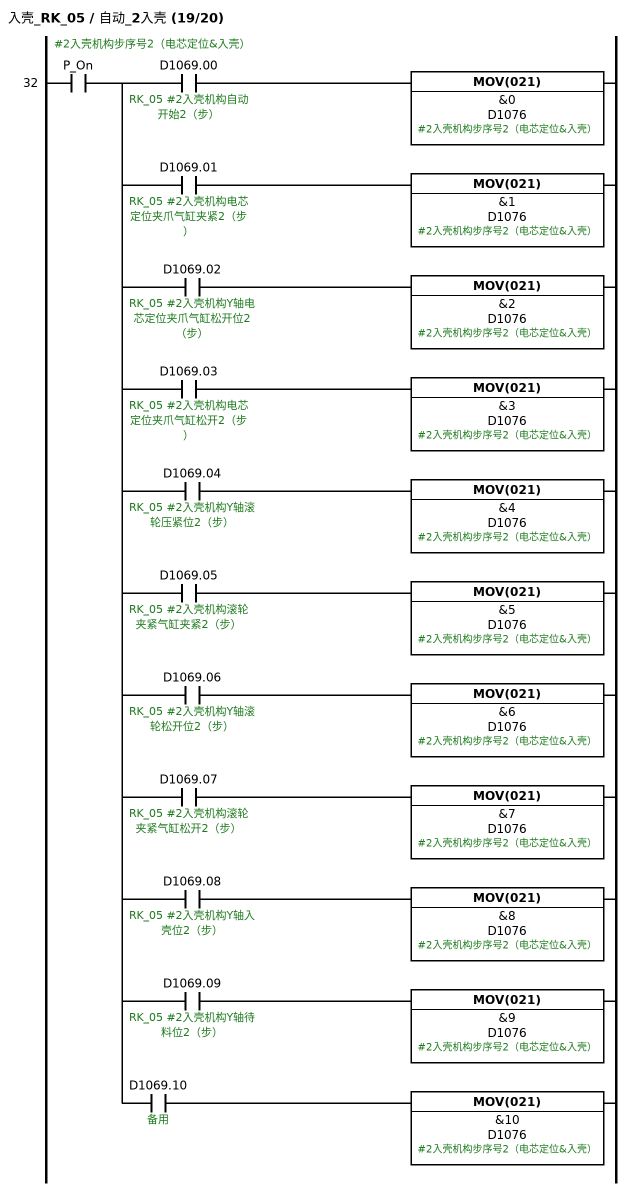
; [picture p480: 入壳_RK_05 / 自动_2入壳, rungs 32-32]
; rung 32: #2入壳机构步序号2（电芯定位&入壳）
LD P_On
OUT TR0
AND D1069.00  ; RK_05 #2入壳机构自动开始2（步）
MOV(021) &0 D1076  ; #2入壳机构步序号2（电芯定位&入壳）
LD TR0
AND D1069.01  ; RK_05 #2入壳机构电芯定位夹爪气缸夹紧2（步）
MOV(021) &1 D1076  ; #2入壳机构步序号2（电芯定位&入壳）
LD TR0
AND D1069.02  ; RK_05 #2入壳机构Y轴电芯定位夹爪气缸松开位2（步）
MOV(021) &2 D1076  ; #2入壳机构步序号2（电芯定位&入壳）
LD TR0
AND D1069.03  ; RK_05 #2入壳机构电芯定位夹爪气缸松开2（步）
MOV(021) &3 D1076  ; #2入壳机构步序号2（电芯定位&入壳）
LD TR0
AND D1069.04  ; RK_05 #2入壳机构Y轴滚轮压紧位2（步）
MOV(021) &4 D1076  ; #2入壳机构步序号2（电芯定位&入壳）
LD TR0
AND D1069.05  ; RK_05 #2入壳机构滚轮夹紧气缸夹紧2（步）
MOV(021) &5 D1076  ; #2入壳机构步序号2（电芯定位&入壳）
LD TR0
AND D1069.06  ; RK_05 #2入壳机构Y轴滚轮松开位2（步）
MOV(021) &6 D1076  ; #2入壳机构步序号2（电芯定位&入壳）
LD TR0
AND D1069.07  ; RK_05 #2入壳机构滚轮夹紧气缸松开2（步）
MOV(021) &7 D1076  ; #2入壳机构步序号2（电芯定位&入壳）
LD TR0
AND D1069.08  ; RK_05 #2入壳机构Y轴入壳位2（步）
MOV(021) &8 D1076  ; #2入壳机构步序号2（电芯定位&入壳）
LD TR0
AND D1069.09  ; RK_05 #2入壳机构Y轴待料位2（步）
MOV(021) &9 D1076  ; #2入壳机构步序号2（电芯定位&入壳）
LD TR0
AND D1069.10  ; 备用
MOV(021) &10 D1076  ; #2入壳机构步序号2（电芯定位&入壳）

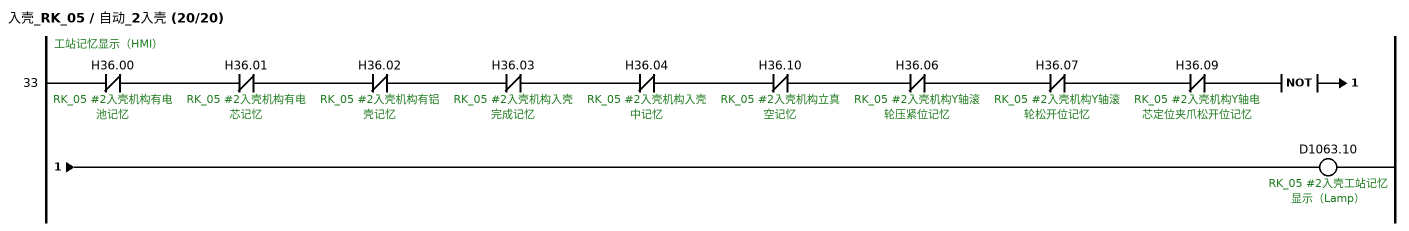
; rung 33: 工站记忆显示（HMI）
LDNOT H36.00  ; RK_05 #2入壳机构有电池记忆
ANDNOT H36.01  ; RK_05 #2入壳机构有电芯记忆
ANDNOT H36.02  ; RK_05 #2入壳机构有铝壳记忆
ANDNOT H36.03  ; RK_05 #2入壳机构入壳完成记忆
ANDNOT H36.04  ; RK_05 #2入壳机构入壳中记忆
ANDNOT H36.10  ; RK_05 #2入壳机构立真空记忆
ANDNOT H36.06  ; RK_05 #2入壳机构Y轴滚轮压紧位记忆
ANDNOT H36.07  ; RK_05 #2入壳机构Y轴滚轮松开位记忆
ANDNOT H36.09  ; RK_05 #2入壳机构Y轴电芯定位夹爪松开位记忆
NOT(520)
OUT D1063.10  ; RK_05 #2入壳工站记忆显示（Lamp）

### Section 复位

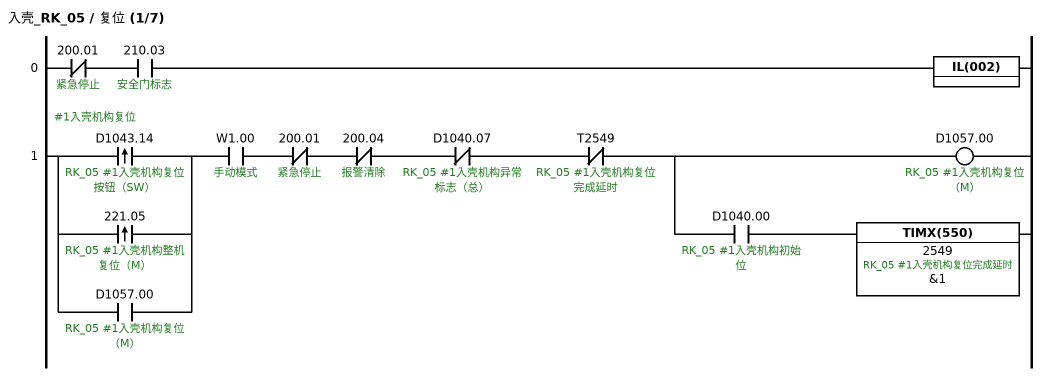
; rung 0
LDNOT 200.01  ; 紧急停止
AND 210.03  ; 安全门标志
IL(002)
; rung 1: #1入壳机构复位
@LD D1043.14  ; RK_05 #1入壳机构复位按钮（SW）
@OR 221.05  ; RK_05 #1入壳机构整机复位（M）
OR D1057.00  ; RK_05 #1入壳机构复位（M）
AND W1.00  ; 手动模式
ANDNOT 200.01  ; 紧急停止
ANDNOT 200.04  ; 报警清除
ANDNOT D1040.07  ; RK_05 #1入壳机构异常标志（总）
ANDNOT T2549  ; RK_05 #1入壳机构复位完成延时
OUT D1057.00  ; RK_05 #1入壳机构复位（M）
AND D1040.00  ; RK_05 #1入壳机构初始位
TIMX(550) 2549 &1  ; RK_05 #1入壳机构复位完成延时

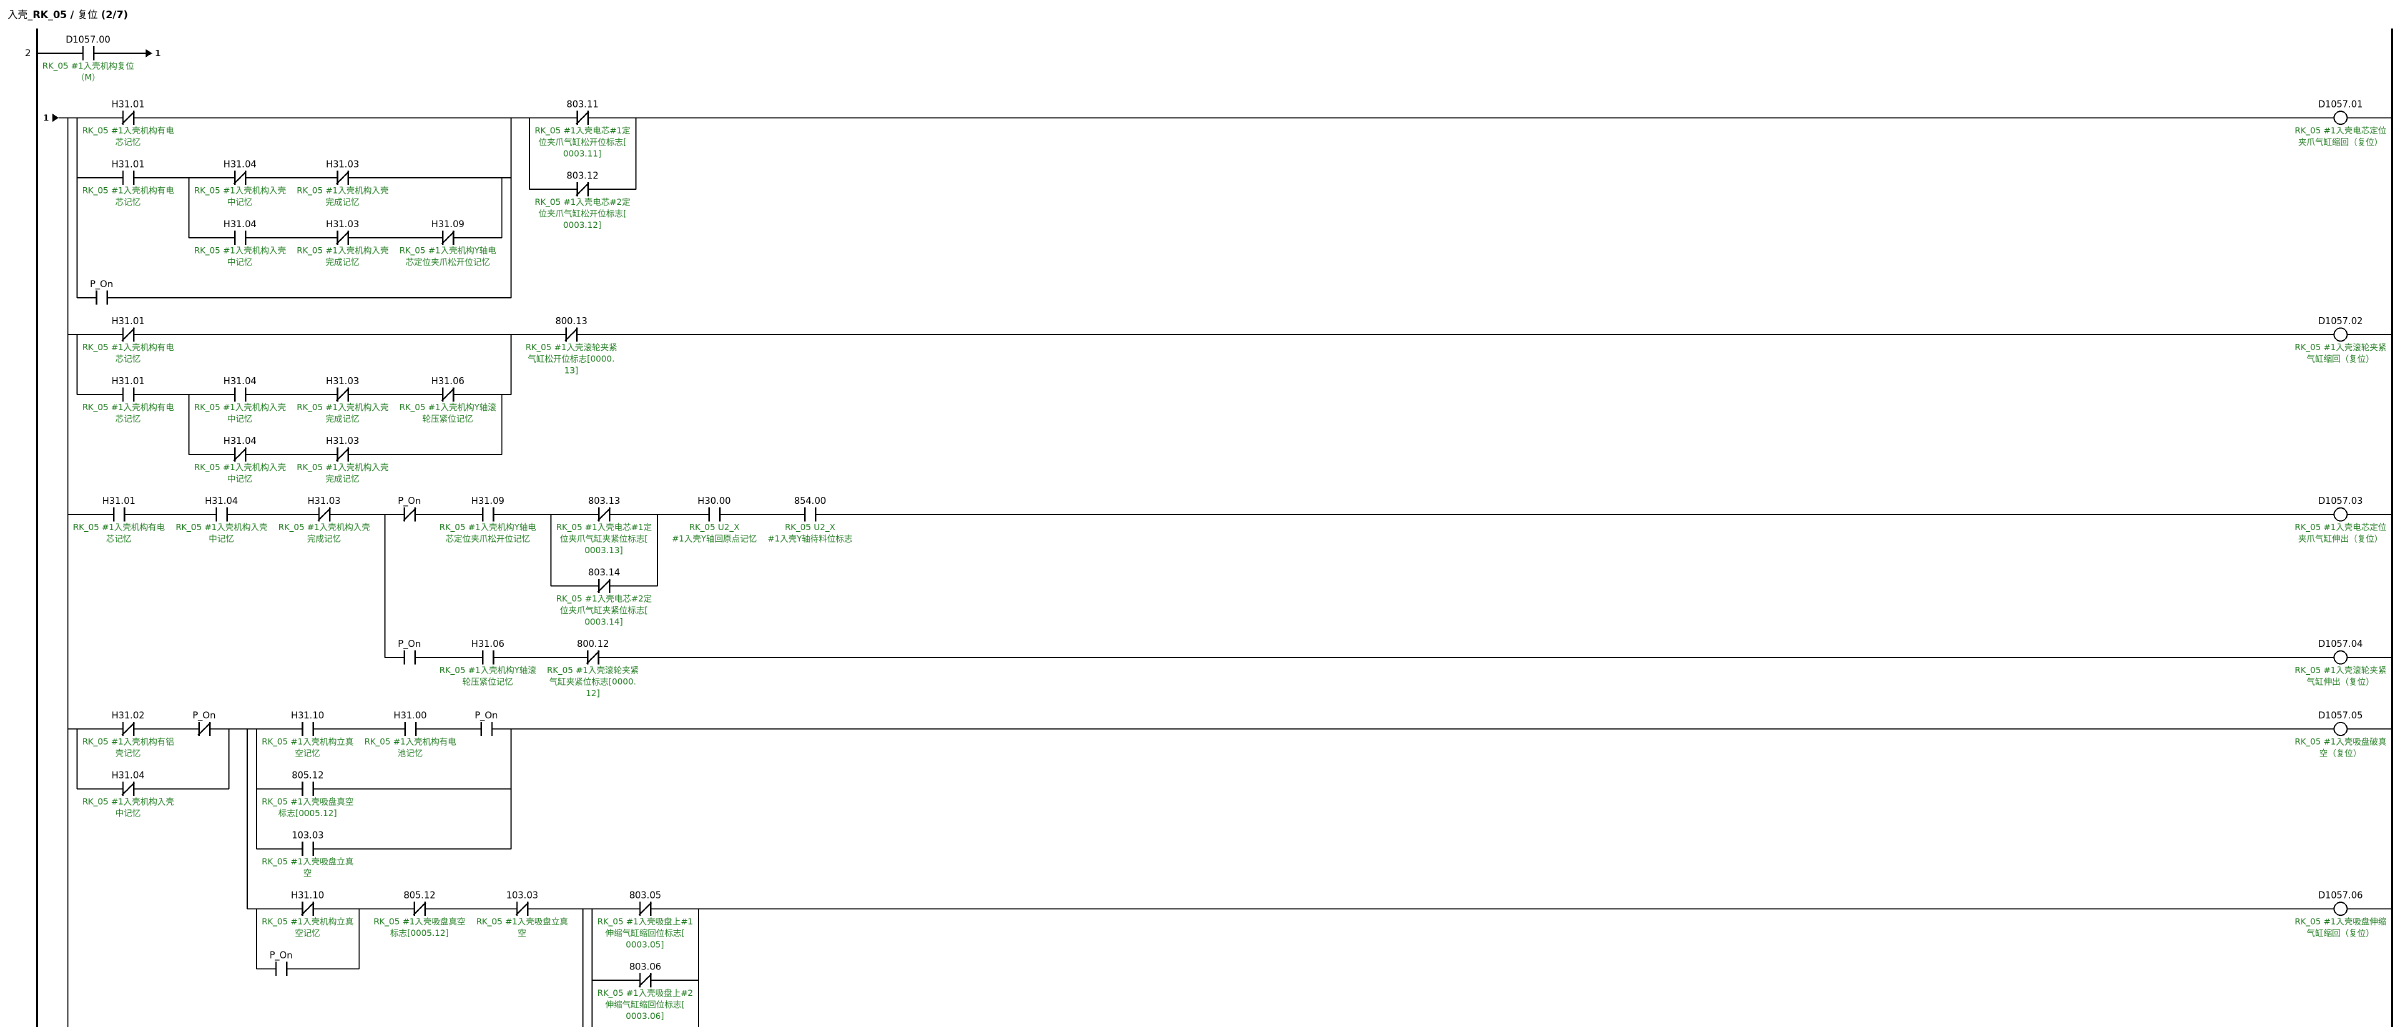

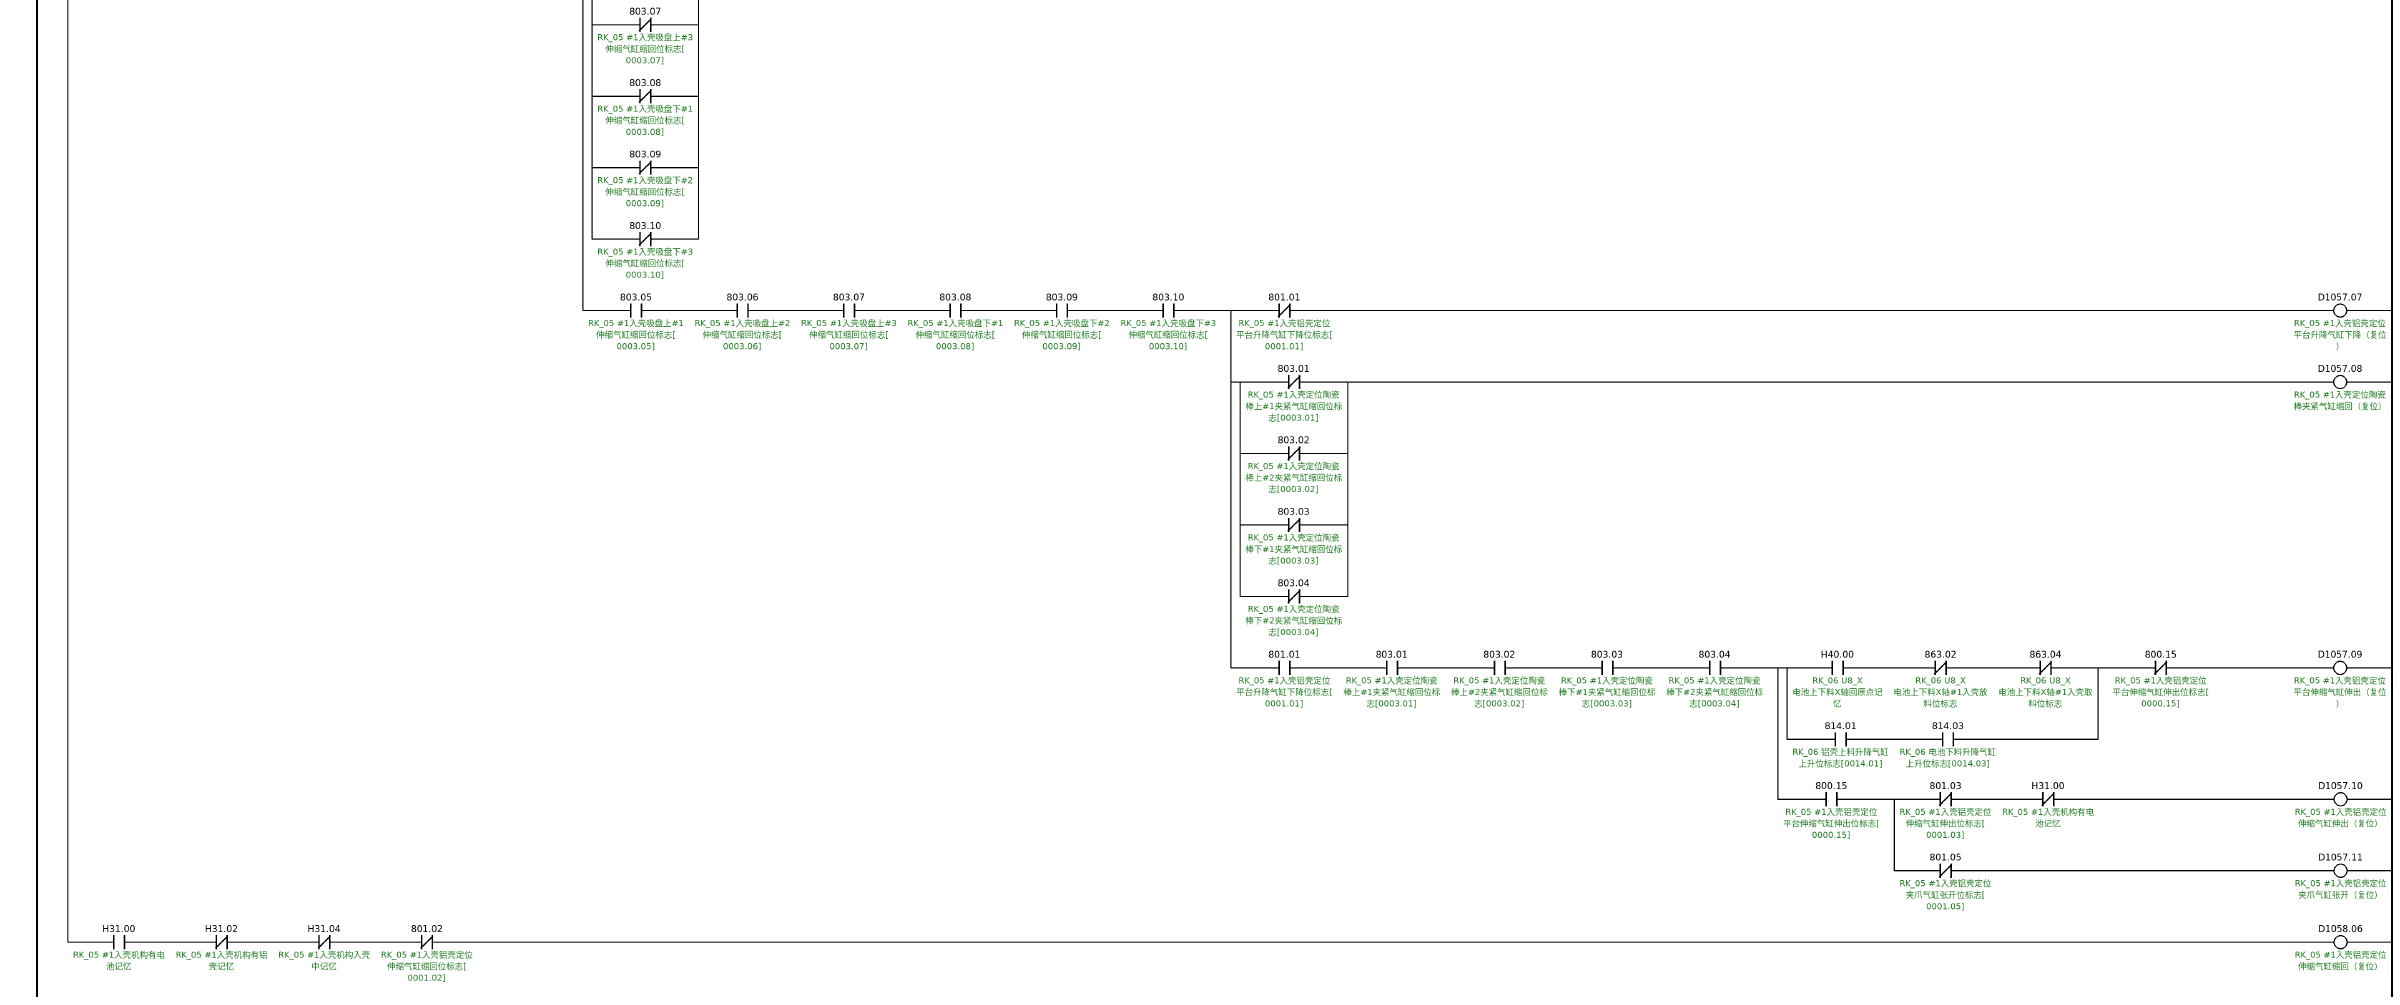
; rung 2
LD D1057.00  ; RK_05 #1入壳机构复位（M）
OUT TR0
LDNOT H31.01  ; RK_05 #1入壳机构有电芯记忆
LD H31.01  ; RK_05 #1入壳机构有电芯记忆
LDNOT H31.04  ; RK_05 #1入壳机构入壳中记忆
ANDNOT H31.03  ; RK_05 #1入壳机构入壳完成记忆
LD H31.04  ; RK_05 #1入壳机构入壳中记忆
ANDNOT H31.03  ; RK_05 #1入壳机构入壳完成记忆
ANDNOT H31.09  ; RK_05 #1入壳机构Y轴电芯定位夹爪松开位记忆
ORLD
ANDLD
ORLD
OR P_On
ANDLD
LDNOT 803.11  ; RK_05 #1入壳电芯#1定位夹爪气缸松开位标志[0003.11]
ORNOT 803.12  ; RK_05 #1入壳电芯#2定位夹爪气缸松开位标志[0003.12]
ANDLD
OUT D1057.01  ; RK_05 #1入壳电芯定位夹爪气缸缩回（复位）
LD TR0
LDNOT H31.01  ; RK_05 #1入壳机构有电芯记忆
LD H31.01  ; RK_05 #1入壳机构有电芯记忆
LD H31.04  ; RK_05 #1入壳机构入壳中记忆
ANDNOT H31.03  ; RK_05 #1入壳机构入壳完成记忆
ANDNOT H31.06  ; RK_05 #1入壳机构Y轴滚轮压紧位记忆
LDNOT H31.04  ; RK_05 #1入壳机构入壳中记忆
ANDNOT H31.03  ; RK_05 #1入壳机构入壳完成记忆
ORLD
ANDLD
ORLD
ANDLD
ANDNOT 800.13  ; RK_05 #1入壳滚轮夹紧气缸松开位标志[0000.13]
OUT D1057.02  ; RK_05 #1入壳滚轮夹紧气缸缩回（复位）
LD TR0
AND H31.01  ; RK_05 #1入壳机构有电芯记忆
AND H31.04  ; RK_05 #1入壳机构入壳中记忆
ANDNOT H31.03  ; RK_05 #1入壳机构入壳完成记忆
OUT TR1
ANDNOT P_On
AND H31.09  ; RK_05 #1入壳机构Y轴电芯定位夹爪松开位记忆
LDNOT 803.13  ; RK_05 #1入壳电芯#1定位夹爪气缸夹紧位标志[0003.13]
ORNOT 803.14  ; RK_05 #1入壳电芯#2定位夹爪气缸夹紧位标志[0003.14]
ANDLD
AND H30.00  ; RK_05 U2_X #1入壳Y轴回原点记忆
AND 854.00  ; RK_05 U2_X #1入壳Y轴待料位标志
OUT D1057.03  ; RK_05 #1入壳电芯定位夹爪气缸伸出（复位）
LD TR1
AND P_On
AND H31.06  ; RK_05 #1入壳机构Y轴滚轮压紧位记忆
ANDNOT 800.12  ; RK_05 #1入壳滚轮夹紧气缸夹紧位标志[0000.12]
OUT D1057.04  ; RK_05 #1入壳滚轮夹紧气缸伸出（复位）
LD TR0
LDNOT H31.02  ; RK_05 #1入壳机构有铝壳记忆
ANDNOT P_On
ORNOT H31.04  ; RK_05 #1入壳机构入壳中记忆
ANDLD
OUT TR1
LD H31.10  ; RK_05 #1入壳机构立真空记忆
AND H31.00  ; RK_05 #1入壳机构有电池记忆
AND P_On
OR 805.12  ; RK_05 #1入壳吸盘真空标志[0005.12]
OR 103.03  ; RK_05 #1入壳吸盘立真空
ANDLD
OUT D1057.05  ; RK_05 #1入壳吸盘破真空（复位）
LD TR1
LDNOT H31.10  ; RK_05 #1入壳机构立真空记忆
OR P_On
ANDLD
ANDNOT 805.12  ; RK_05 #1入壳吸盘真空标志[0005.12]
ANDNOT 103.03  ; RK_05 #1入壳吸盘立真空
OUT TR1
LDNOT 803.05  ; RK_05 #1入壳吸盘上#1伸缩气缸缩回位标志[0003.05]
ORNOT 803.06  ; RK_05 #1入壳吸盘上#2伸缩气缸缩回位标志[0003.06]
ORNOT 803.07  ; RK_05 #1入壳吸盘上#3伸缩气缸缩回位标志[0003.07]
ORNOT 803.08  ; RK_05 #1入壳吸盘下#1伸缩气缸缩回位标志[0003.08]
ORNOT 803.09  ; RK_05 #1入壳吸盘下#2伸缩气缸缩回位标志[0003.09]
ORNOT 803.10  ; RK_05 #1入壳吸盘下#3伸缩气缸缩回位标志[0003.10]
ANDLD
OUT D1057.06  ; RK_05 #1入壳吸盘伸缩气缸缩回（复位）
LD TR1
AND 803.05  ; RK_05 #1入壳吸盘上#1伸缩气缸缩回位标志[0003.05]
AND 803.06  ; RK_05 #1入壳吸盘上#2伸缩气缸缩回位标志[0003.06]
AND 803.07  ; RK_05 #1入壳吸盘上#3伸缩气缸缩回位标志[0003.07]
AND 803.08  ; RK_05 #1入壳吸盘下#1伸缩气缸缩回位标志[0003.08]
AND 803.09  ; RK_05 #1入壳吸盘下#2伸缩气缸缩回位标志[0003.09]
AND 803.10  ; RK_05 #1入壳吸盘下#3伸缩气缸缩回位标志[0003.10]
OUT TR1
ANDNOT 801.01  ; RK_05 #1入壳铝壳定位平台升降气缸下降位标志[0001.01]
OUT D1057.07  ; RK_05 #1入壳铝壳定位平台升降气缸下降（复位）
LD TR1
LDNOT 803.01  ; RK_05 #1入壳定位陶瓷棒上#1夹紧气缸缩回位标志[0003.01]
ORNOT 803.02  ; RK_05 #1入壳定位陶瓷棒上#2夹紧气缸缩回位标志[0003.02]
ORNOT 803.03  ; RK_05 #1入壳定位陶瓷棒下#1夹紧气缸缩回位标志[0003.03]
ORNOT 803.04  ; RK_05 #1入壳定位陶瓷棒下#2夹紧气缸缩回位标志[0003.04]
ANDLD
OUT D1057.08  ; RK_05 #1入壳定位陶瓷棒夹紧气缸缩回（复位）
LD TR1
AND 801.01  ; RK_05 #1入壳铝壳定位平台升降气缸下降位标志[0001.01]
AND 803.01  ; RK_05 #1入壳定位陶瓷棒上#1夹紧气缸缩回位标志[0003.01]
AND 803.02  ; RK_05 #1入壳定位陶瓷棒上#2夹紧气缸缩回位标志[0003.02]
AND 803.03  ; RK_05 #1入壳定位陶瓷棒下#1夹紧气缸缩回位标志[0003.03]
AND 803.04  ; RK_05 #1入壳定位陶瓷棒下#2夹紧气缸缩回位标志[0003.04]
OUT TR1
LD H40.00  ; RK_06 U8_X 电池上下料X轴回原点记忆
ANDNOT 863.02  ; RK_06 U8_X 电池上下料X轴#1入壳放料位标志
ANDNOT 863.04  ; RK_06 U8_X 电池上下料X轴#1入壳取料位标志
LD 814.01  ; RK_06 铝壳上料升降气缸上升位标志[0014.01]
AND 814.03  ; RK_06 电池下料升降气缸上升位标志[0014.03]
ORLD
ANDLD
ANDNOT 800.15  ; RK_05 #1入壳铝壳定位平台伸缩气缸伸出位标志[0000.15]
OUT D1057.09  ; RK_05 #1入壳铝壳定位平台伸缩气缸伸出（复位）
LD TR1
AND 800.15  ; RK_05 #1入壳铝壳定位平台伸缩气缸伸出位标志[0000.15]
OUT TR1
ANDNOT 801.03  ; RK_05 #1入壳铝壳定位伸缩气缸伸出位标志[0001.03]
ANDNOT H31.00  ; RK_05 #1入壳机构有电池记忆
OUT D1057.10  ; RK_05 #1入壳铝壳定位伸缩气缸伸出（复位）
LD TR1
ANDNOT 801.05  ; RK_05 #1入壳铝壳定位夹爪气缸张开位标志[0001.05]
OUT D1057.11  ; RK_05 #1入壳铝壳定位夹爪气缸张开（复位）
LD TR0
AND H31.00  ; RK_05 #1入壳机构有电池记忆
ANDNOT H31.02  ; RK_05 #1入壳机构有铝壳记忆
ANDNOT H31.04  ; RK_05 #1入壳机构入壳中记忆
ANDNOT 801.02  ; RK_05 #1入壳铝壳定位伸缩气缸缩回位标志[0001.02]
OUT D1058.06  ; RK_05 #1入壳铝壳定位伸缩气缸缩回（复位）

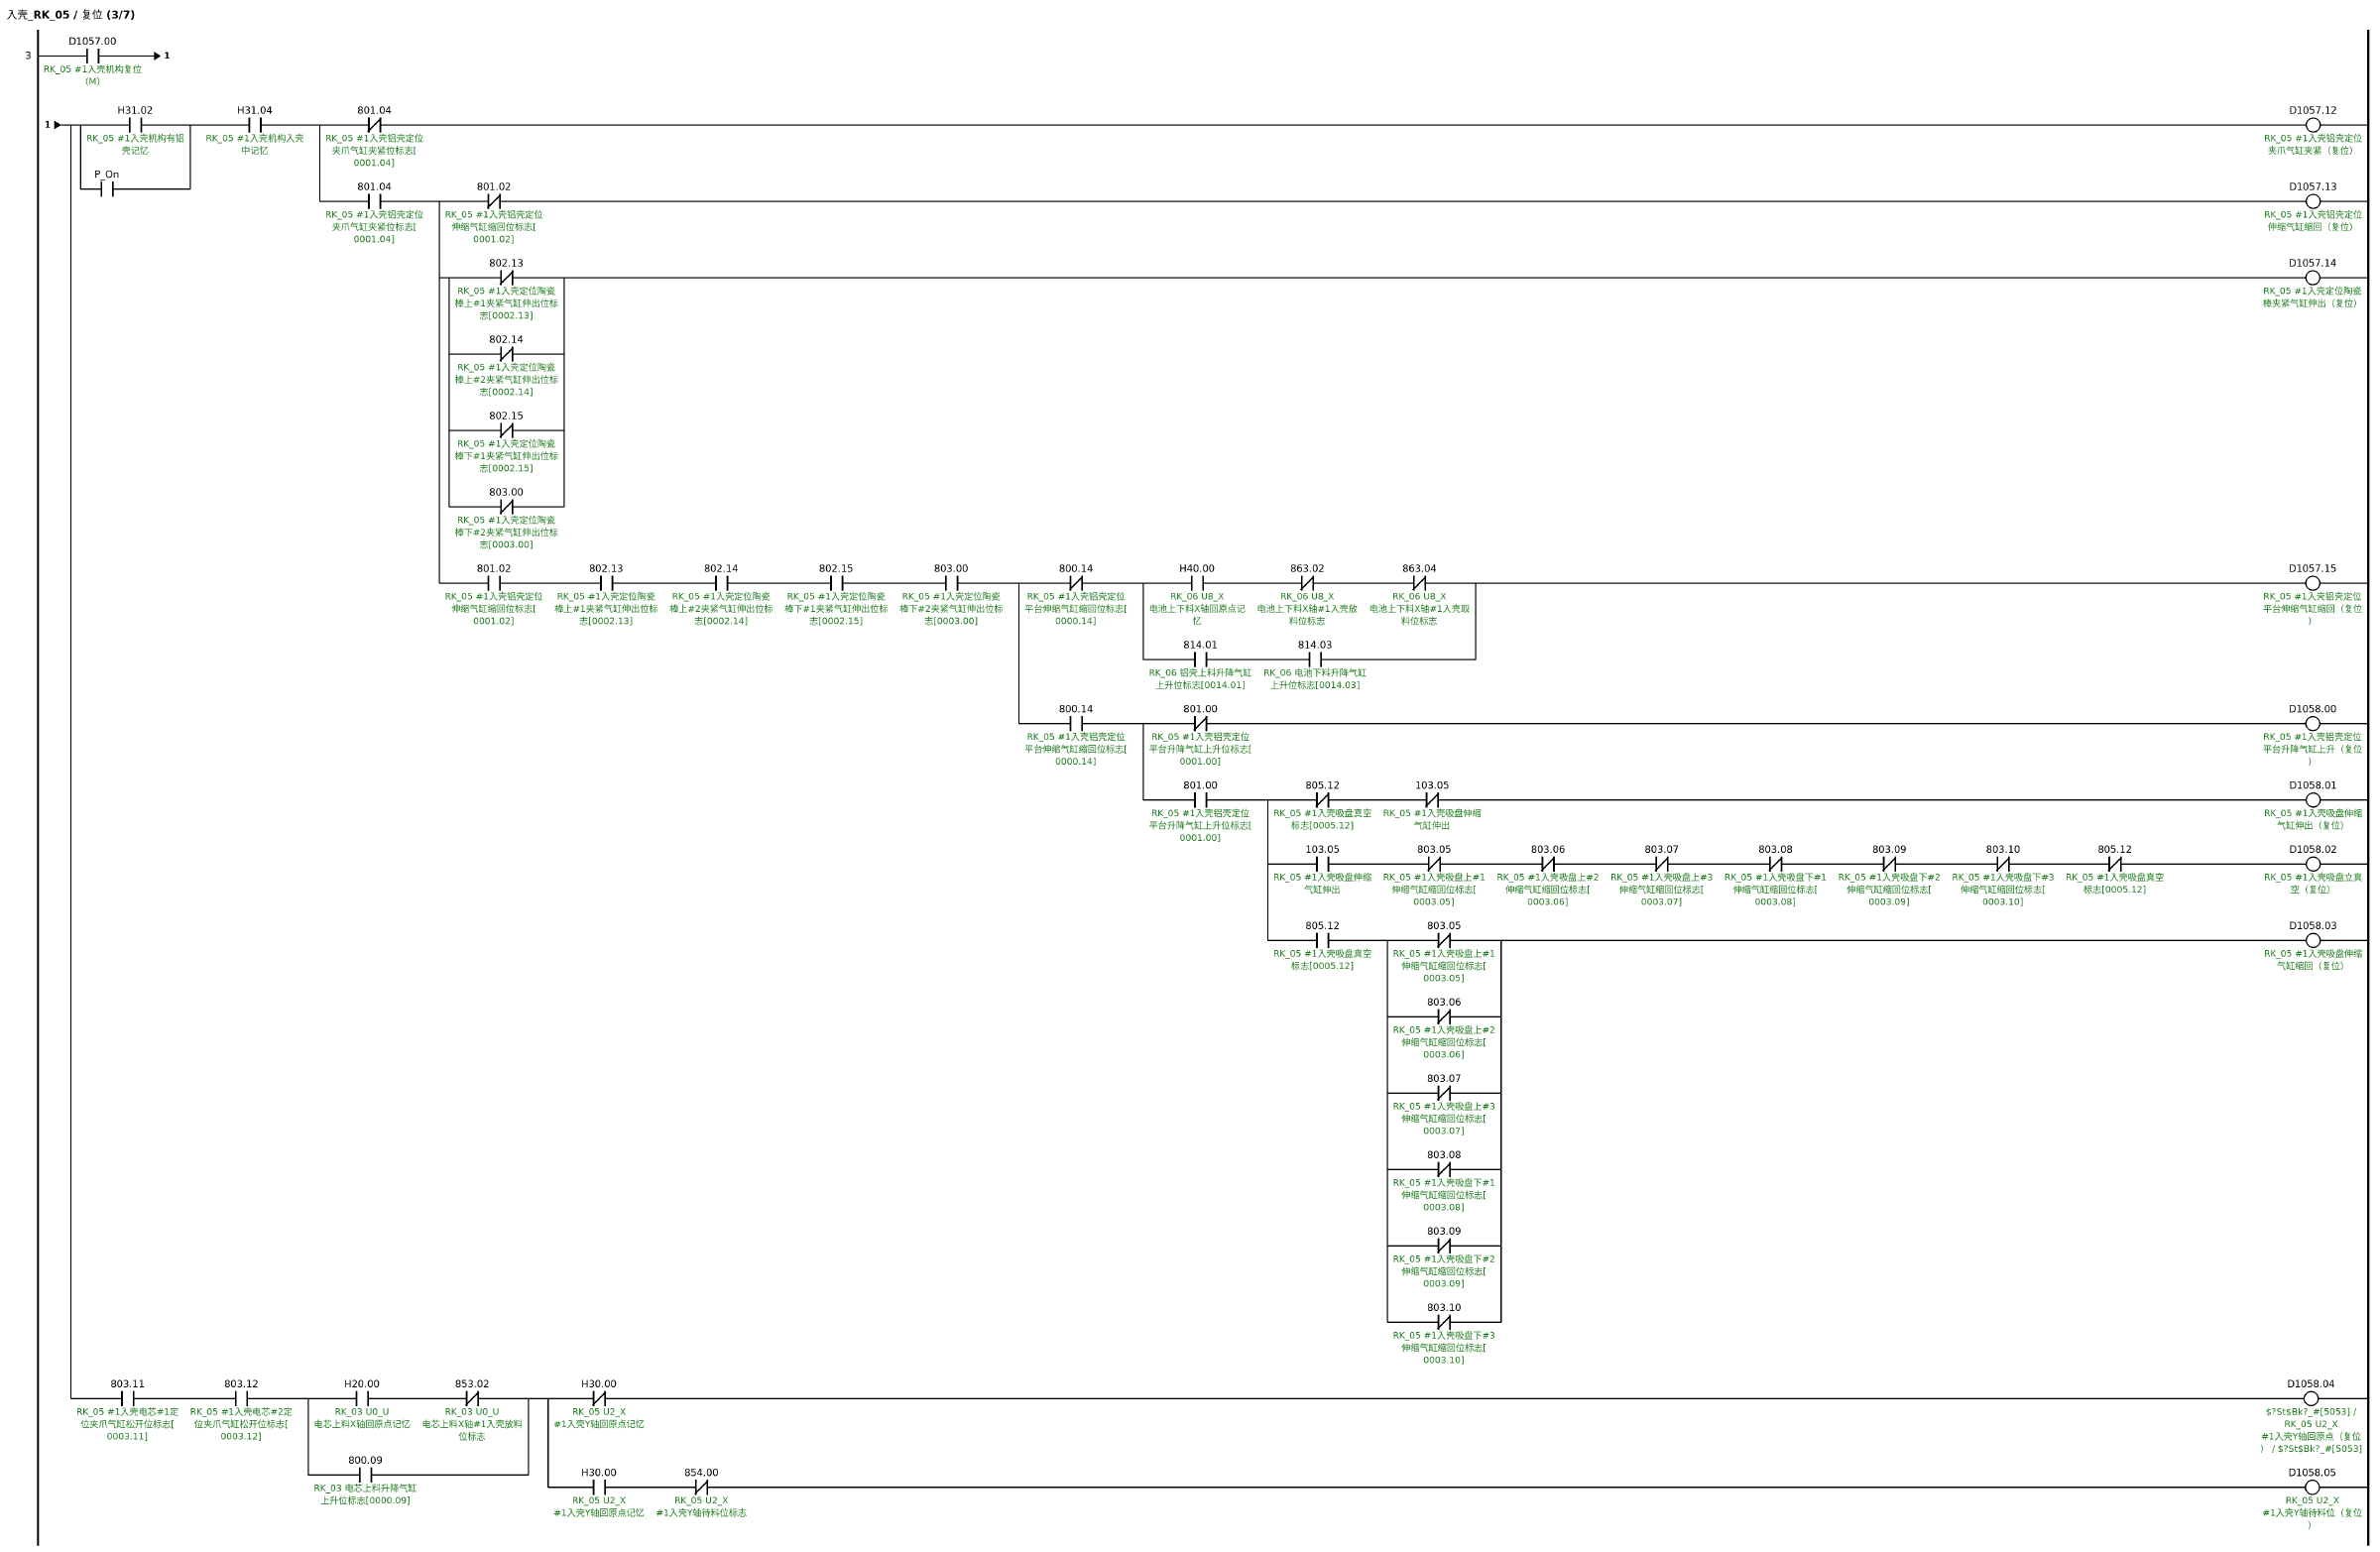
; rung 3
LD D1057.00  ; RK_05 #1入壳机构复位（M）
OUT TR0
LD H31.02  ; RK_05 #1入壳机构有铝壳记忆
OR P_On
ANDLD
AND H31.04  ; RK_05 #1入壳机构入壳中记忆
OUT TR1
ANDNOT 801.04  ; RK_05 #1入壳铝壳定位夹爪气缸夹紧位标志[0001.04]
OUT D1057.12  ; RK_05 #1入壳铝壳定位夹爪气缸夹紧（复位）
LD TR1
AND 801.04  ; RK_05 #1入壳铝壳定位夹爪气缸夹紧位标志[0001.04]
OUT TR1
ANDNOT 801.02  ; RK_05 #1入壳铝壳定位伸缩气缸缩回位标志[0001.02]
OUT D1057.13  ; RK_05 #1入壳铝壳定位伸缩气缸缩回（复位）
LD TR1
LDNOT 802.13  ; RK_05 #1入壳定位陶瓷棒上#1夹紧气缸伸出位标志[0002.13]
ORNOT 802.14  ; RK_05 #1入壳定位陶瓷棒上#2夹紧气缸伸出位标志[0002.14]
ORNOT 802.15  ; RK_05 #1入壳定位陶瓷棒下#1夹紧气缸伸出位标志[0002.15]
ORNOT 803.00  ; RK_05 #1入壳定位陶瓷棒下#2夹紧气缸伸出位标志[0003.00]
ANDLD
OUT D1057.14  ; RK_05 #1入壳定位陶瓷棒夹紧气缸伸出（复位）
LD TR1
AND 801.02  ; RK_05 #1入壳铝壳定位伸缩气缸缩回位标志[0001.02]
AND 802.13  ; RK_05 #1入壳定位陶瓷棒上#1夹紧气缸伸出位标志[0002.13]
AND 802.14  ; RK_05 #1入壳定位陶瓷棒上#2夹紧气缸伸出位标志[0002.14]
AND 802.15  ; RK_05 #1入壳定位陶瓷棒下#1夹紧气缸伸出位标志[0002.15]
AND 803.00  ; RK_05 #1入壳定位陶瓷棒下#2夹紧气缸伸出位标志[0003.00]
OUT TR1
ANDNOT 800.14  ; RK_05 #1入壳铝壳定位平台伸缩气缸缩回位标志[0000.14]
LD H40.00  ; RK_06 U8_X 电池上下料X轴回原点记忆
ANDNOT 863.02  ; RK_06 U8_X 电池上下料X轴#1入壳放料位标志
ANDNOT 863.04  ; RK_06 U8_X 电池上下料X轴#1入壳取料位标志
LD 814.01  ; RK_06 铝壳上料升降气缸上升位标志[0014.01]
AND 814.03  ; RK_06 电池下料升降气缸上升位标志[0014.03]
ORLD
ANDLD
OUT D1057.15  ; RK_05 #1入壳铝壳定位平台伸缩气缸缩回（复位）
LD TR1
AND 800.14  ; RK_05 #1入壳铝壳定位平台伸缩气缸缩回位标志[0000.14]
OUT TR1
ANDNOT 801.00  ; RK_05 #1入壳铝壳定位平台升降气缸上升位标志[0001.00]
OUT D1058.00  ; RK_05 #1入壳铝壳定位平台升降气缸上升（复位）
LD TR1
AND 801.00  ; RK_05 #1入壳铝壳定位平台升降气缸上升位标志[0001.00]
OUT TR1
ANDNOT 805.12  ; RK_05 #1入壳吸盘真空标志[0005.12]
ANDNOT 103.05  ; RK_05 #1入壳吸盘伸缩气缸伸出
OUT D1058.01  ; RK_05 #1入壳吸盘伸缩气缸伸出（复位）
LD TR1
AND 103.05  ; RK_05 #1入壳吸盘伸缩气缸伸出
ANDNOT 803.05  ; RK_05 #1入壳吸盘上#1伸缩气缸缩回位标志[0003.05]
ANDNOT 803.06  ; RK_05 #1入壳吸盘上#2伸缩气缸缩回位标志[0003.06]
ANDNOT 803.07  ; RK_05 #1入壳吸盘上#3伸缩气缸缩回位标志[0003.07]
ANDNOT 803.08  ; RK_05 #1入壳吸盘下#1伸缩气缸缩回位标志[0003.08]
ANDNOT 803.09  ; RK_05 #1入壳吸盘下#2伸缩气缸缩回位标志[0003.09]
ANDNOT 803.10  ; RK_05 #1入壳吸盘下#3伸缩气缸缩回位标志[0003.10]
ANDNOT 805.12  ; RK_05 #1入壳吸盘真空标志[0005.12]
OUT D1058.02  ; RK_05 #1入壳吸盘立真空（复位）
LD TR1
AND 805.12  ; RK_05 #1入壳吸盘真空标志[0005.12]
LDNOT 803.05  ; RK_05 #1入壳吸盘上#1伸缩气缸缩回位标志[0003.05]
ORNOT 803.06  ; RK_05 #1入壳吸盘上#2伸缩气缸缩回位标志[0003.06]
ORNOT 803.07  ; RK_05 #1入壳吸盘上#3伸缩气缸缩回位标志[0003.07]
ORNOT 803.08  ; RK_05 #1入壳吸盘下#1伸缩气缸缩回位标志[0003.08]
ORNOT 803.09  ; RK_05 #1入壳吸盘下#2伸缩气缸缩回位标志[0003.09]
ORNOT 803.10  ; RK_05 #1入壳吸盘下#3伸缩气缸缩回位标志[0003.10]
ANDLD
OUT D1058.03  ; RK_05 #1入壳吸盘伸缩气缸缩回（复位）
LD TR0
AND 803.11  ; RK_05 #1入壳电芯#1定位夹爪气缸松开位标志[0003.11]
AND 803.12  ; RK_05 #1入壳电芯#2定位夹爪气缸松开位标志[0003.12]
LD H20.00  ; RK_03 U0_U 电芯上料X轴回原点记忆
ANDNOT 853.02  ; RK_03 U0_U 电芯上料X轴#1入壳放料位标志
OR 800.09  ; RK_03 电芯上料升降气缸上升位标志[0000.09]
ANDLD
OUT TR0
ANDNOT H30.00  ; RK_05 U2_X #1入壳Y轴回原点记忆
OUT D1058.04  ; $?St$Bk?_#[5053] / RK_05 U2_X #1入壳Y轴回原点（复位） / $?St$Bk?_#[5053]
LD TR0
AND H30.00  ; RK_05 U2_X #1入壳Y轴回原点记忆
ANDNOT 854.00  ; RK_05 U2_X #1入壳Y轴待料位标志
OUT D1058.05  ; RK_05 U2_X #1入壳Y轴待料位（复位）

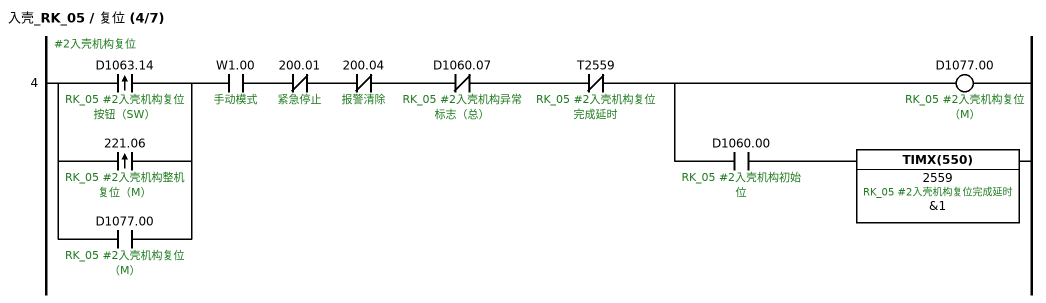
; rung 4: #2入壳机构复位
@LD D1063.14  ; RK_05 #2入壳机构复位按钮（SW）
@OR 221.06  ; RK_05 #2入壳机构整机复位（M）
OR D1077.00  ; RK_05 #2入壳机构复位（M）
AND W1.00  ; 手动模式
ANDNOT 200.01  ; 紧急停止
ANDNOT 200.04  ; 报警清除
ANDNOT D1060.07  ; RK_05 #2入壳机构异常标志（总）
ANDNOT T2559  ; RK_05 #2入壳机构复位完成延时
OUT D1077.00  ; RK_05 #2入壳机构复位（M）
AND D1060.00  ; RK_05 #2入壳机构初始位
TIMX(550) 2559 &1  ; RK_05 #2入壳机构复位完成延时

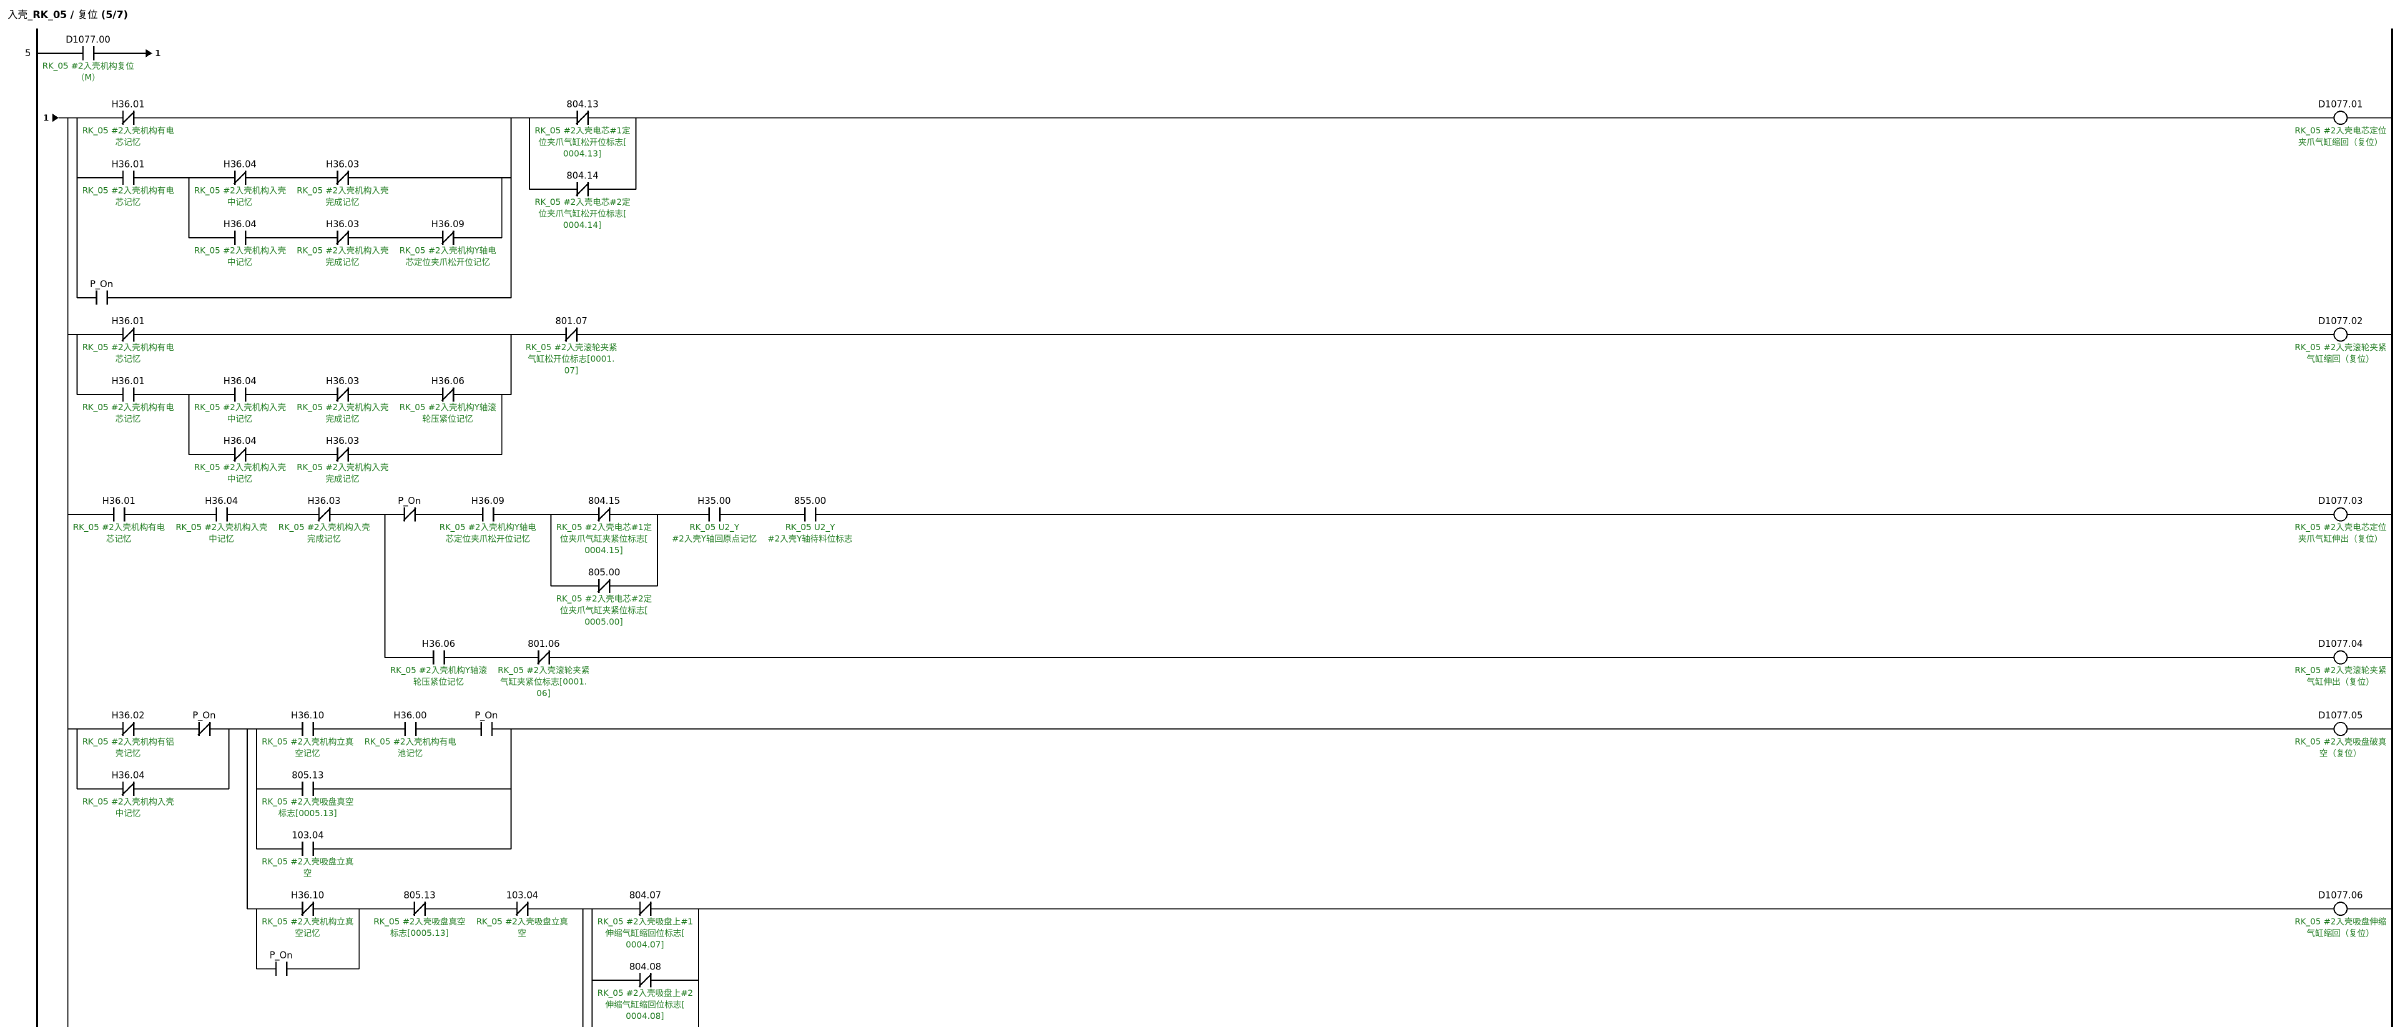

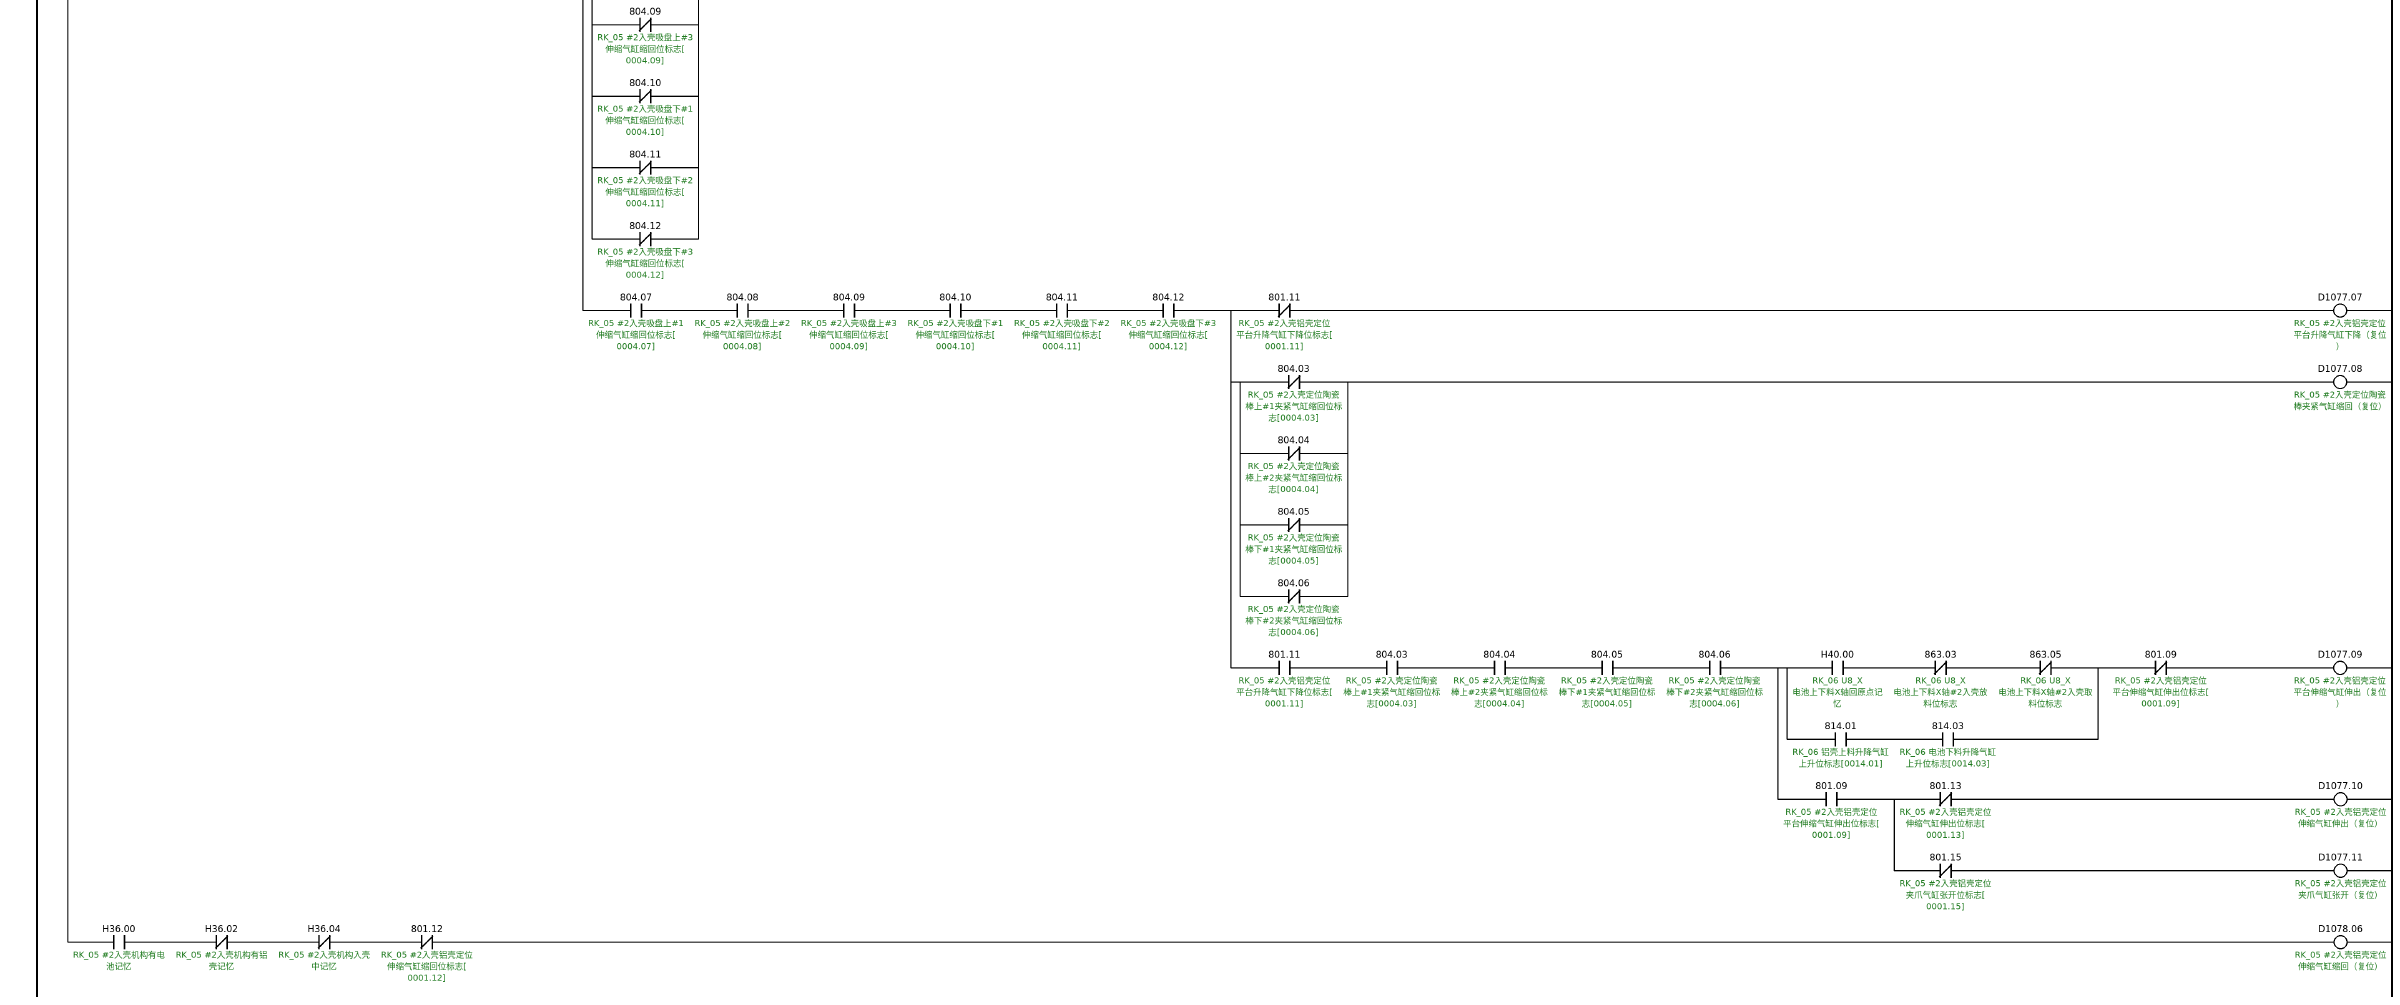
; rung 5
LD D1077.00  ; RK_05 #2入壳机构复位（M）
OUT TR0
LDNOT H36.01  ; RK_05 #2入壳机构有电芯记忆
LD H36.01  ; RK_05 #2入壳机构有电芯记忆
LDNOT H36.04  ; RK_05 #2入壳机构入壳中记忆
ANDNOT H36.03  ; RK_05 #2入壳机构入壳完成记忆
LD H36.04  ; RK_05 #2入壳机构入壳中记忆
ANDNOT H36.03  ; RK_05 #2入壳机构入壳完成记忆
ANDNOT H36.09  ; RK_05 #2入壳机构Y轴电芯定位夹爪松开位记忆
ORLD
ANDLD
ORLD
OR P_On
ANDLD
LDNOT 804.13  ; RK_05 #2入壳电芯#1定位夹爪气缸松开位标志[0004.13]
ORNOT 804.14  ; RK_05 #2入壳电芯#2定位夹爪气缸松开位标志[0004.14]
ANDLD
OUT D1077.01  ; RK_05 #2入壳电芯定位夹爪气缸缩回（复位）
LD TR0
LDNOT H36.01  ; RK_05 #2入壳机构有电芯记忆
LD H36.01  ; RK_05 #2入壳机构有电芯记忆
LD H36.04  ; RK_05 #2入壳机构入壳中记忆
ANDNOT H36.03  ; RK_05 #2入壳机构入壳完成记忆
ANDNOT H36.06  ; RK_05 #2入壳机构Y轴滚轮压紧位记忆
LDNOT H36.04  ; RK_05 #2入壳机构入壳中记忆
ANDNOT H36.03  ; RK_05 #2入壳机构入壳完成记忆
ORLD
ANDLD
ORLD
ANDLD
ANDNOT 801.07  ; RK_05 #2入壳滚轮夹紧气缸松开位标志[0001.07]
OUT D1077.02  ; RK_05 #2入壳滚轮夹紧气缸缩回（复位）
LD TR0
AND H36.01  ; RK_05 #2入壳机构有电芯记忆
AND H36.04  ; RK_05 #2入壳机构入壳中记忆
ANDNOT H36.03  ; RK_05 #2入壳机构入壳完成记忆
OUT TR1
ANDNOT P_On
AND H36.09  ; RK_05 #2入壳机构Y轴电芯定位夹爪松开位记忆
LDNOT 804.15  ; RK_05 #2入壳电芯#1定位夹爪气缸夹紧位标志[0004.15]
ORNOT 805.00  ; RK_05 #2入壳电芯#2定位夹爪气缸夹紧位标志[0005.00]
ANDLD
AND H35.00  ; RK_05 U2_Y #2入壳Y轴回原点记忆
AND 855.00  ; RK_05 U2_Y #2入壳Y轴待料位标志
OUT D1077.03  ; RK_05 #2入壳电芯定位夹爪气缸伸出（复位）
LD TR1
AND H36.06  ; RK_05 #2入壳机构Y轴滚轮压紧位记忆
ANDNOT 801.06  ; RK_05 #2入壳滚轮夹紧气缸夹紧位标志[0001.06]
OUT D1077.04  ; RK_05 #2入壳滚轮夹紧气缸伸出（复位）
LD TR0
LDNOT H36.02  ; RK_05 #2入壳机构有铝壳记忆
ANDNOT P_On
ORNOT H36.04  ; RK_05 #2入壳机构入壳中记忆
ANDLD
OUT TR1
LD H36.10  ; RK_05 #2入壳机构立真空记忆
AND H36.00  ; RK_05 #2入壳机构有电池记忆
AND P_On
OR 805.13  ; RK_05 #2入壳吸盘真空标志[0005.13]
OR 103.04  ; RK_05 #2入壳吸盘立真空
ANDLD
OUT D1077.05  ; RK_05 #2入壳吸盘破真空（复位）
LD TR1
LDNOT H36.10  ; RK_05 #2入壳机构立真空记忆
OR P_On
ANDLD
ANDNOT 805.13  ; RK_05 #2入壳吸盘真空标志[0005.13]
ANDNOT 103.04  ; RK_05 #2入壳吸盘立真空
OUT TR1
LDNOT 804.07  ; RK_05 #2入壳吸盘上#1伸缩气缸缩回位标志[0004.07]
ORNOT 804.08  ; RK_05 #2入壳吸盘上#2伸缩气缸缩回位标志[0004.08]
ORNOT 804.09  ; RK_05 #2入壳吸盘上#3伸缩气缸缩回位标志[0004.09]
ORNOT 804.10  ; RK_05 #2入壳吸盘下#1伸缩气缸缩回位标志[0004.10]
ORNOT 804.11  ; RK_05 #2入壳吸盘下#2伸缩气缸缩回位标志[0004.11]
ORNOT 804.12  ; RK_05 #2入壳吸盘下#3伸缩气缸缩回位标志[0004.12]
ANDLD
OUT D1077.06  ; RK_05 #2入壳吸盘伸缩气缸缩回（复位）
LD TR1
AND 804.07  ; RK_05 #2入壳吸盘上#1伸缩气缸缩回位标志[0004.07]
AND 804.08  ; RK_05 #2入壳吸盘上#2伸缩气缸缩回位标志[0004.08]
AND 804.09  ; RK_05 #2入壳吸盘上#3伸缩气缸缩回位标志[0004.09]
AND 804.10  ; RK_05 #2入壳吸盘下#1伸缩气缸缩回位标志[0004.10]
AND 804.11  ; RK_05 #2入壳吸盘下#2伸缩气缸缩回位标志[0004.11]
AND 804.12  ; RK_05 #2入壳吸盘下#3伸缩气缸缩回位标志[0004.12]
OUT TR1
ANDNOT 801.11  ; RK_05 #2入壳铝壳定位平台升降气缸下降位标志[0001.11]
OUT D1077.07  ; RK_05 #2入壳铝壳定位平台升降气缸下降（复位）
LD TR1
LDNOT 804.03  ; RK_05 #2入壳定位陶瓷棒上#1夹紧气缸缩回位标志[0004.03]
ORNOT 804.04  ; RK_05 #2入壳定位陶瓷棒上#2夹紧气缸缩回位标志[0004.04]
ORNOT 804.05  ; RK_05 #2入壳定位陶瓷棒下#1夹紧气缸缩回位标志[0004.05]
ORNOT 804.06  ; RK_05 #2入壳定位陶瓷棒下#2夹紧气缸缩回位标志[0004.06]
ANDLD
OUT D1077.08  ; RK_05 #2入壳定位陶瓷棒夹紧气缸缩回（复位）
LD TR1
AND 801.11  ; RK_05 #2入壳铝壳定位平台升降气缸下降位标志[0001.11]
AND 804.03  ; RK_05 #2入壳定位陶瓷棒上#1夹紧气缸缩回位标志[0004.03]
AND 804.04  ; RK_05 #2入壳定位陶瓷棒上#2夹紧气缸缩回位标志[0004.04]
AND 804.05  ; RK_05 #2入壳定位陶瓷棒下#1夹紧气缸缩回位标志[0004.05]
AND 804.06  ; RK_05 #2入壳定位陶瓷棒下#2夹紧气缸缩回位标志[0004.06]
OUT TR1
LD H40.00  ; RK_06 U8_X 电池上下料X轴回原点记忆
ANDNOT 863.03  ; RK_06 U8_X 电池上下料X轴#2入壳放料位标志
ANDNOT 863.05  ; RK_06 U8_X 电池上下料X轴#2入壳取料位标志
LD 814.01  ; RK_06 铝壳上料升降气缸上升位标志[0014.01]
AND 814.03  ; RK_06 电池下料升降气缸上升位标志[0014.03]
ORLD
ANDLD
ANDNOT 801.09  ; RK_05 #2入壳铝壳定位平台伸缩气缸伸出位标志[0001.09]
OUT D1077.09  ; RK_05 #2入壳铝壳定位平台伸缩气缸伸出（复位）
LD TR1
AND 801.09  ; RK_05 #2入壳铝壳定位平台伸缩气缸伸出位标志[0001.09]
OUT TR1
ANDNOT 801.13  ; RK_05 #2入壳铝壳定位伸缩气缸伸出位标志[0001.13]
OUT D1077.10  ; RK_05 #2入壳铝壳定位伸缩气缸伸出（复位）
LD TR1
ANDNOT 801.15  ; RK_05 #2入壳铝壳定位夹爪气缸张开位标志[0001.15]
OUT D1077.11  ; RK_05 #2入壳铝壳定位夹爪气缸张开（复位）
LD TR0
AND H36.00  ; RK_05 #2入壳机构有电池记忆
ANDNOT H36.02  ; RK_05 #2入壳机构有铝壳记忆
ANDNOT H36.04  ; RK_05 #2入壳机构入壳中记忆
ANDNOT 801.12  ; RK_05 #2入壳铝壳定位伸缩气缸缩回位标志[0001.12]
OUT D1078.06  ; RK_05 #2入壳铝壳定位伸缩气缸缩回（复位）

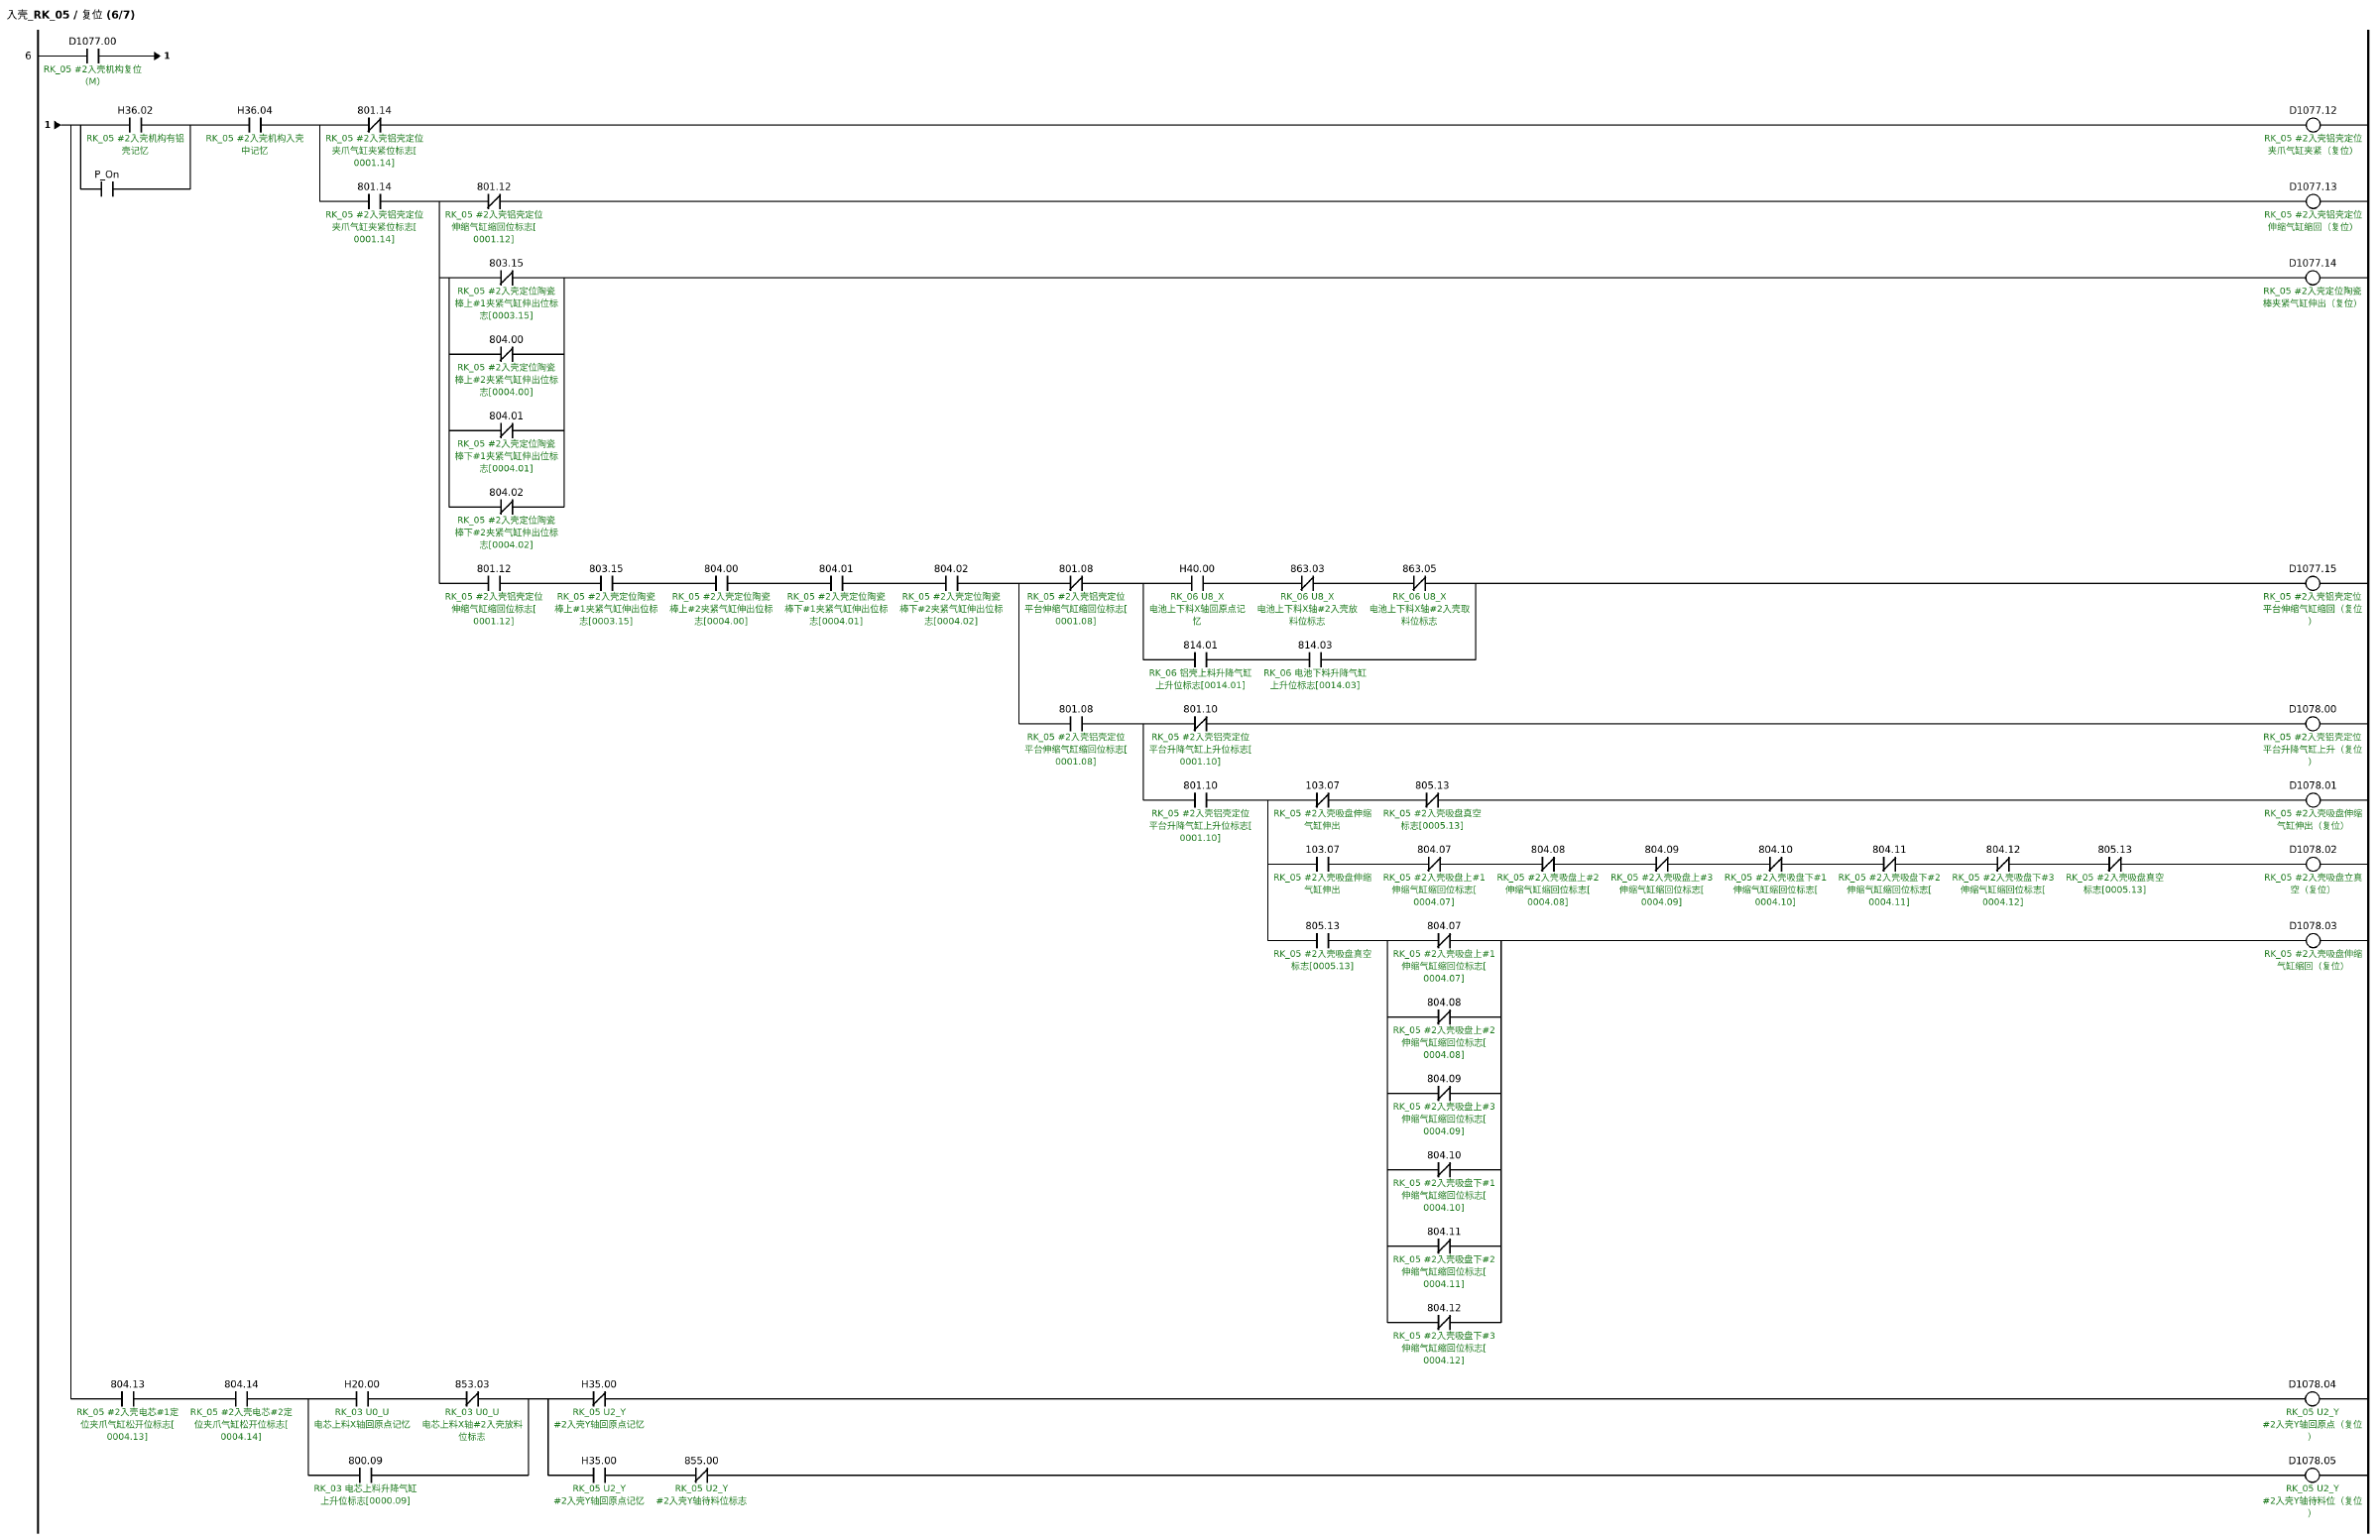
; rung 6
LD D1077.00  ; RK_05 #2入壳机构复位（M）
OUT TR0
LD H36.02  ; RK_05 #2入壳机构有铝壳记忆
OR P_On
ANDLD
AND H36.04  ; RK_05 #2入壳机构入壳中记忆
OUT TR1
ANDNOT 801.14  ; RK_05 #2入壳铝壳定位夹爪气缸夹紧位标志[0001.14]
OUT D1077.12  ; RK_05 #2入壳铝壳定位夹爪气缸夹紧（复位）
LD TR1
AND 801.14  ; RK_05 #2入壳铝壳定位夹爪气缸夹紧位标志[0001.14]
OUT TR1
ANDNOT 801.12  ; RK_05 #2入壳铝壳定位伸缩气缸缩回位标志[0001.12]
OUT D1077.13  ; RK_05 #2入壳铝壳定位伸缩气缸缩回（复位）
LD TR1
LDNOT 803.15  ; RK_05 #2入壳定位陶瓷棒上#1夹紧气缸伸出位标志[0003.15]
ORNOT 804.00  ; RK_05 #2入壳定位陶瓷棒上#2夹紧气缸伸出位标志[0004.00]
ORNOT 804.01  ; RK_05 #2入壳定位陶瓷棒下#1夹紧气缸伸出位标志[0004.01]
ORNOT 804.02  ; RK_05 #2入壳定位陶瓷棒下#2夹紧气缸伸出位标志[0004.02]
ANDLD
OUT D1077.14  ; RK_05 #2入壳定位陶瓷棒夹紧气缸伸出（复位）
LD TR1
AND 801.12  ; RK_05 #2入壳铝壳定位伸缩气缸缩回位标志[0001.12]
AND 803.15  ; RK_05 #2入壳定位陶瓷棒上#1夹紧气缸伸出位标志[0003.15]
AND 804.00  ; RK_05 #2入壳定位陶瓷棒上#2夹紧气缸伸出位标志[0004.00]
AND 804.01  ; RK_05 #2入壳定位陶瓷棒下#1夹紧气缸伸出位标志[0004.01]
AND 804.02  ; RK_05 #2入壳定位陶瓷棒下#2夹紧气缸伸出位标志[0004.02]
OUT TR1
ANDNOT 801.08  ; RK_05 #2入壳铝壳定位平台伸缩气缸缩回位标志[0001.08]
LD H40.00  ; RK_06 U8_X 电池上下料X轴回原点记忆
ANDNOT 863.03  ; RK_06 U8_X 电池上下料X轴#2入壳放料位标志
ANDNOT 863.05  ; RK_06 U8_X 电池上下料X轴#2入壳取料位标志
LD 814.01  ; RK_06 铝壳上料升降气缸上升位标志[0014.01]
AND 814.03  ; RK_06 电池下料升降气缸上升位标志[0014.03]
ORLD
ANDLD
OUT D1077.15  ; RK_05 #2入壳铝壳定位平台伸缩气缸缩回（复位）
LD TR1
AND 801.08  ; RK_05 #2入壳铝壳定位平台伸缩气缸缩回位标志[0001.08]
OUT TR1
ANDNOT 801.10  ; RK_05 #2入壳铝壳定位平台升降气缸上升位标志[0001.10]
OUT D1078.00  ; RK_05 #2入壳铝壳定位平台升降气缸上升（复位）
LD TR1
AND 801.10  ; RK_05 #2入壳铝壳定位平台升降气缸上升位标志[0001.10]
OUT TR1
ANDNOT 103.07  ; RK_05 #2入壳吸盘伸缩气缸伸出
ANDNOT 805.13  ; RK_05 #2入壳吸盘真空标志[0005.13]  // 20181116新增
OUT D1078.01  ; RK_05 #2入壳吸盘伸缩气缸伸出（复位）
LD TR1
AND 103.07  ; RK_05 #2入壳吸盘伸缩气缸伸出
ANDNOT 804.07  ; RK_05 #2入壳吸盘上#1伸缩气缸缩回位标志[0004.07]
ANDNOT 804.08  ; RK_05 #2入壳吸盘上#2伸缩气缸缩回位标志[0004.08]
ANDNOT 804.09  ; RK_05 #2入壳吸盘上#3伸缩气缸缩回位标志[0004.09]
ANDNOT 804.10  ; RK_05 #2入壳吸盘下#1伸缩气缸缩回位标志[0004.10]
ANDNOT 804.11  ; RK_05 #2入壳吸盘下#2伸缩气缸缩回位标志[0004.11]
ANDNOT 804.12  ; RK_05 #2入壳吸盘下#3伸缩气缸缩回位标志[0004.12]
ANDNOT 805.13  ; RK_05 #2入壳吸盘真空标志[0005.13]
OUT D1078.02  ; RK_05 #2入壳吸盘立真空（复位）
LD TR1
AND 805.13  ; RK_05 #2入壳吸盘真空标志[0005.13]
LDNOT 804.07  ; RK_05 #2入壳吸盘上#1伸缩气缸缩回位标志[0004.07]
ORNOT 804.08  ; RK_05 #2入壳吸盘上#2伸缩气缸缩回位标志[0004.08]
ORNOT 804.09  ; RK_05 #2入壳吸盘上#3伸缩气缸缩回位标志[0004.09]
ORNOT 804.10  ; RK_05 #2入壳吸盘下#1伸缩气缸缩回位标志[0004.10]
ORNOT 804.11  ; RK_05 #2入壳吸盘下#2伸缩气缸缩回位标志[0004.11]
ORNOT 804.12  ; RK_05 #2入壳吸盘下#3伸缩气缸缩回位标志[0004.12]
ANDLD
OUT D1078.03  ; RK_05 #2入壳吸盘伸缩气缸缩回（复位）
LD TR0
AND 804.13  ; RK_05 #2入壳电芯#1定位夹爪气缸松开位标志[0004.13]
AND 804.14  ; RK_05 #2入壳电芯#2定位夹爪气缸松开位标志[0004.14]
LD H20.00  ; RK_03 U0_U 电芯上料X轴回原点记忆
ANDNOT 853.03  ; RK_03 U0_U 电芯上料X轴#2入壳放料位标志
OR 800.09  ; RK_03 电芯上料升降气缸上升位标志[0000.09]
ANDLD
OUT TR0
ANDNOT H35.00  ; RK_05 U2_Y #2入壳Y轴回原点记忆
OUT D1078.04  ; RK_05 U2_Y #2入壳Y轴回原点（复位）
LD TR0
AND H35.00  ; RK_05 U2_Y #2入壳Y轴回原点记忆
ANDNOT 855.00  ; RK_05 U2_Y #2入壳Y轴待料位标志
OUT D1078.05  ; RK_05 U2_Y #2入壳Y轴待料位（复位）

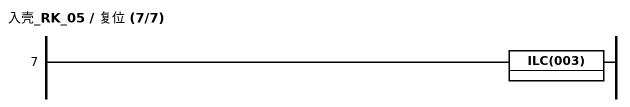
; rung 7
ILC(003)

### Section 指示灯

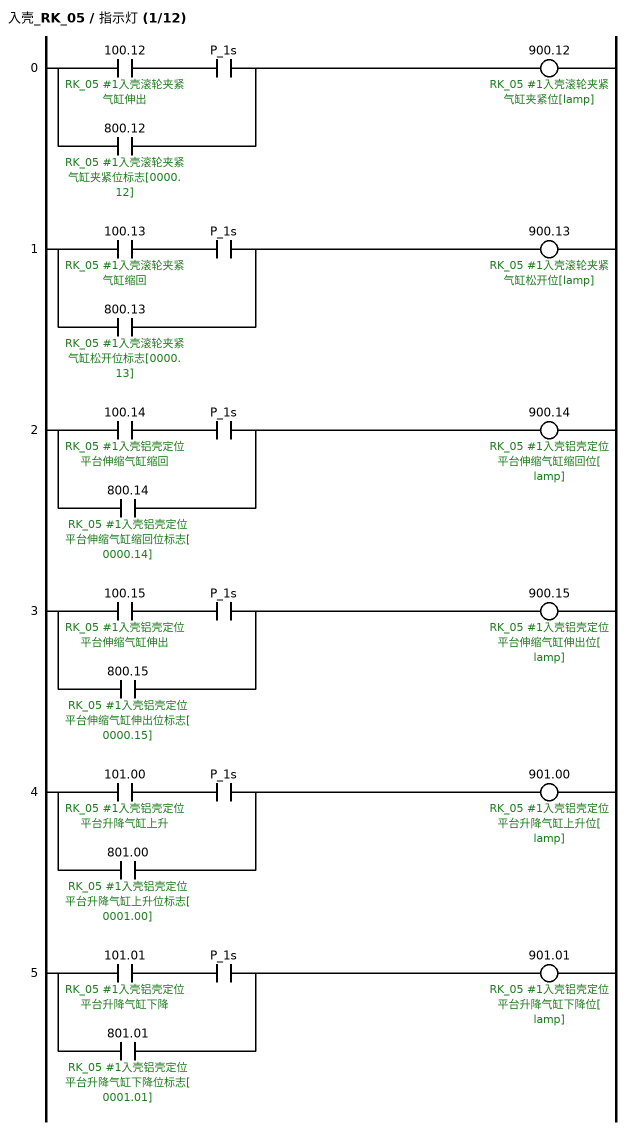
; rung 0
LD 100.12  ; RK_05 #1入壳滚轮夹紧气缸伸出
AND P_1s
OR 800.12  ; RK_05 #1入壳滚轮夹紧气缸夹紧位标志[0000.12]
OUT 900.12  ; RK_05 #1入壳滚轮夹紧气缸夹紧位[lamp]
; rung 1
LD 100.13  ; RK_05 #1入壳滚轮夹紧气缸缩回
AND P_1s
OR 800.13  ; RK_05 #1入壳滚轮夹紧气缸松开位标志[0000.13]
OUT 900.13  ; RK_05 #1入壳滚轮夹紧气缸松开位[lamp]
; rung 2
LD 100.14  ; RK_05 #1入壳铝壳定位平台伸缩气缸缩回
AND P_1s
OR 800.14  ; RK_05 #1入壳铝壳定位平台伸缩气缸缩回位标志[0000.14]
OUT 900.14  ; RK_05 #1入壳铝壳定位平台伸缩气缸缩回位[lamp]
; rung 3
LD 100.15  ; RK_05 #1入壳铝壳定位平台伸缩气缸伸出
AND P_1s
OR 800.15  ; RK_05 #1入壳铝壳定位平台伸缩气缸伸出位标志[0000.15]
OUT 900.15  ; RK_05 #1入壳铝壳定位平台伸缩气缸伸出位[lamp]
; rung 4
LD 101.00  ; RK_05 #1入壳铝壳定位平台升降气缸上升
AND P_1s
OR 801.00  ; RK_05 #1入壳铝壳定位平台升降气缸上升位标志[0001.00]
OUT 901.00  ; RK_05 #1入壳铝壳定位平台升降气缸上升位[lamp]
; rung 5
LD 101.01  ; RK_05 #1入壳铝壳定位平台升降气缸下降
AND P_1s
OR 801.01  ; RK_05 #1入壳铝壳定位平台升降气缸下降位标志[0001.01]
OUT 901.01  ; RK_05 #1入壳铝壳定位平台升降气缸下降位[lamp]

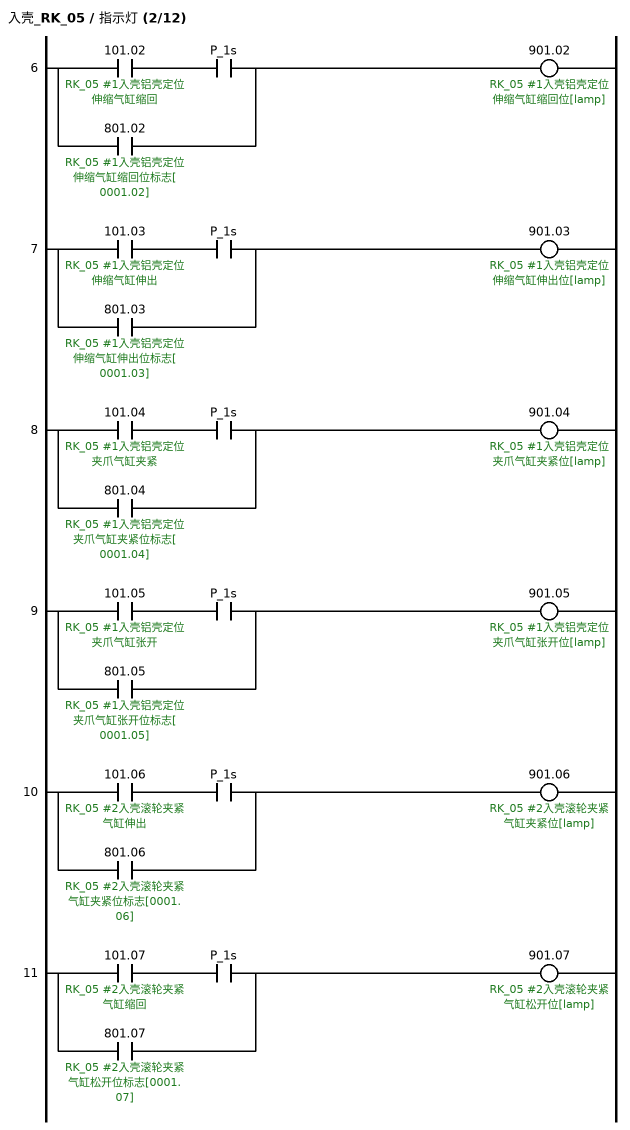
; rung 6
LD 101.02  ; RK_05 #1入壳铝壳定位伸缩气缸缩回
AND P_1s
OR 801.02  ; RK_05 #1入壳铝壳定位伸缩气缸缩回位标志[0001.02]
OUT 901.02  ; RK_05 #1入壳铝壳定位伸缩气缸缩回位[lamp]
; rung 7
LD 101.03  ; RK_05 #1入壳铝壳定位伸缩气缸伸出
AND P_1s
OR 801.03  ; RK_05 #1入壳铝壳定位伸缩气缸伸出位标志[0001.03]
OUT 901.03  ; RK_05 #1入壳铝壳定位伸缩气缸伸出位[lamp]
; rung 8
LD 101.04  ; RK_05 #1入壳铝壳定位夹爪气缸夹紧
AND P_1s
OR 801.04  ; RK_05 #1入壳铝壳定位夹爪气缸夹紧位标志[0001.04]
OUT 901.04  ; RK_05 #1入壳铝壳定位夹爪气缸夹紧位[lamp]
; rung 9
LD 101.05  ; RK_05 #1入壳铝壳定位夹爪气缸张开
AND P_1s
OR 801.05  ; RK_05 #1入壳铝壳定位夹爪气缸张开位标志[0001.05]
OUT 901.05  ; RK_05 #1入壳铝壳定位夹爪气缸张开位[lamp]
; rung 10
LD 101.06  ; RK_05 #2入壳滚轮夹紧气缸伸出
AND P_1s
OR 801.06  ; RK_05 #2入壳滚轮夹紧气缸夹紧位标志[0001.06]
OUT 901.06  ; RK_05 #2入壳滚轮夹紧气缸夹紧位[lamp]
; rung 11
LD 101.07  ; RK_05 #2入壳滚轮夹紧气缸缩回
AND P_1s
OR 801.07  ; RK_05 #2入壳滚轮夹紧气缸松开位标志[0001.07]
OUT 901.07  ; RK_05 #2入壳滚轮夹紧气缸松开位[lamp]

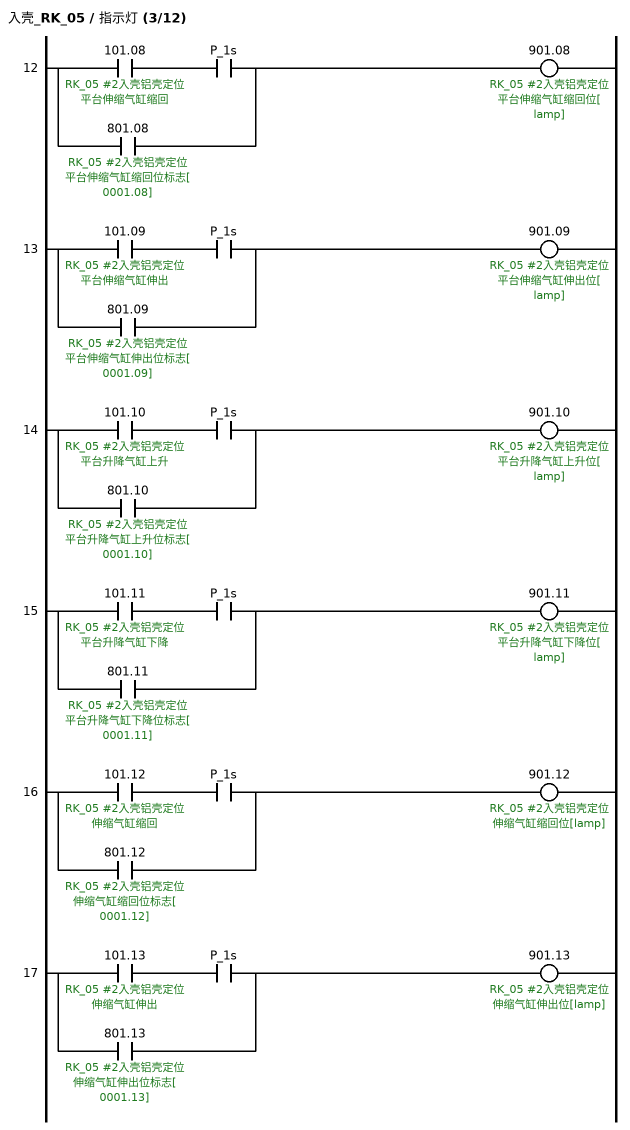
; rung 12
LD 101.08  ; RK_05 #2入壳铝壳定位平台伸缩气缸缩回
AND P_1s
OR 801.08  ; RK_05 #2入壳铝壳定位平台伸缩气缸缩回位标志[0001.08]
OUT 901.08  ; RK_05 #2入壳铝壳定位平台伸缩气缸缩回位[lamp]
; rung 13
LD 101.09  ; RK_05 #2入壳铝壳定位平台伸缩气缸伸出
AND P_1s
OR 801.09  ; RK_05 #2入壳铝壳定位平台伸缩气缸伸出位标志[0001.09]
OUT 901.09  ; RK_05 #2入壳铝壳定位平台伸缩气缸伸出位[lamp]
; rung 14
LD 101.10  ; RK_05 #2入壳铝壳定位平台升降气缸上升
AND P_1s
OR 801.10  ; RK_05 #2入壳铝壳定位平台升降气缸上升位标志[0001.10]
OUT 901.10  ; RK_05 #2入壳铝壳定位平台升降气缸上升位[lamp]
; rung 15
LD 101.11  ; RK_05 #2入壳铝壳定位平台升降气缸下降
AND P_1s
OR 801.11  ; RK_05 #2入壳铝壳定位平台升降气缸下降位标志[0001.11]
OUT 901.11  ; RK_05 #2入壳铝壳定位平台升降气缸下降位[lamp]
; rung 16
LD 101.12  ; RK_05 #2入壳铝壳定位伸缩气缸缩回
AND P_1s
OR 801.12  ; RK_05 #2入壳铝壳定位伸缩气缸缩回位标志[0001.12]
OUT 901.12  ; RK_05 #2入壳铝壳定位伸缩气缸缩回位[lamp]
; rung 17
LD 101.13  ; RK_05 #2入壳铝壳定位伸缩气缸伸出
AND P_1s
OR 801.13  ; RK_05 #2入壳铝壳定位伸缩气缸伸出位标志[0001.13]
OUT 901.13  ; RK_05 #2入壳铝壳定位伸缩气缸伸出位[lamp]

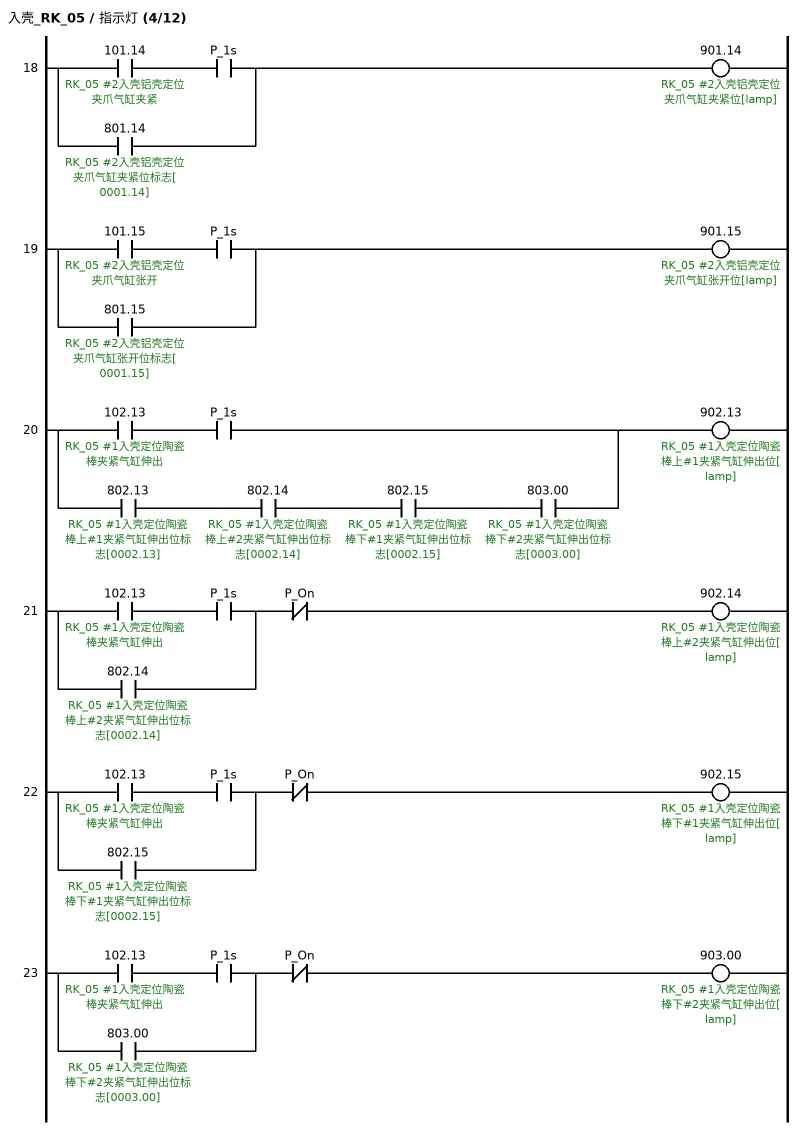
; rung 18
LD 101.14  ; RK_05 #2入壳铝壳定位夹爪气缸夹紧
AND P_1s
OR 801.14  ; RK_05 #2入壳铝壳定位夹爪气缸夹紧位标志[0001.14]
OUT 901.14  ; RK_05 #2入壳铝壳定位夹爪气缸夹紧位[lamp]
; rung 19
LD 101.15  ; RK_05 #2入壳铝壳定位夹爪气缸张开
AND P_1s
OR 801.15  ; RK_05 #2入壳铝壳定位夹爪气缸张开位标志[0001.15]
OUT 901.15  ; RK_05 #2入壳铝壳定位夹爪气缸张开位[lamp]
; rung 20
LD 102.13  ; RK_05 #1入壳定位陶瓷棒夹紧气缸伸出
AND P_1s
LD 802.13  ; RK_05 #1入壳定位陶瓷棒上#1夹紧气缸伸出位标志[0002.13]
AND 802.14  ; RK_05 #1入壳定位陶瓷棒上#2夹紧气缸伸出位标志[0002.14]
AND 802.15  ; RK_05 #1入壳定位陶瓷棒下#1夹紧气缸伸出位标志[0002.15]
AND 803.00  ; RK_05 #1入壳定位陶瓷棒下#2夹紧气缸伸出位标志[0003.00]
ORLD
OUT 902.13  ; RK_05 #1入壳定位陶瓷棒上#1夹紧气缸伸出位[lamp]
; rung 21
LD 102.13  ; RK_05 #1入壳定位陶瓷棒夹紧气缸伸出
AND P_1s
OR 802.14  ; RK_05 #1入壳定位陶瓷棒上#2夹紧气缸伸出位标志[0002.14]
ANDNOT P_On
OUT 902.14  ; RK_05 #1入壳定位陶瓷棒上#2夹紧气缸伸出位[lamp]
; rung 22
LD 102.13  ; RK_05 #1入壳定位陶瓷棒夹紧气缸伸出
AND P_1s
OR 802.15  ; RK_05 #1入壳定位陶瓷棒下#1夹紧气缸伸出位标志[0002.15]
ANDNOT P_On
OUT 902.15  ; RK_05 #1入壳定位陶瓷棒下#1夹紧气缸伸出位[lamp]
; rung 23
LD 102.13  ; RK_05 #1入壳定位陶瓷棒夹紧气缸伸出
AND P_1s
OR 803.00  ; RK_05 #1入壳定位陶瓷棒下#2夹紧气缸伸出位标志[0003.00]
ANDNOT P_On
OUT 903.00  ; RK_05 #1入壳定位陶瓷棒下#2夹紧气缸伸出位[lamp]

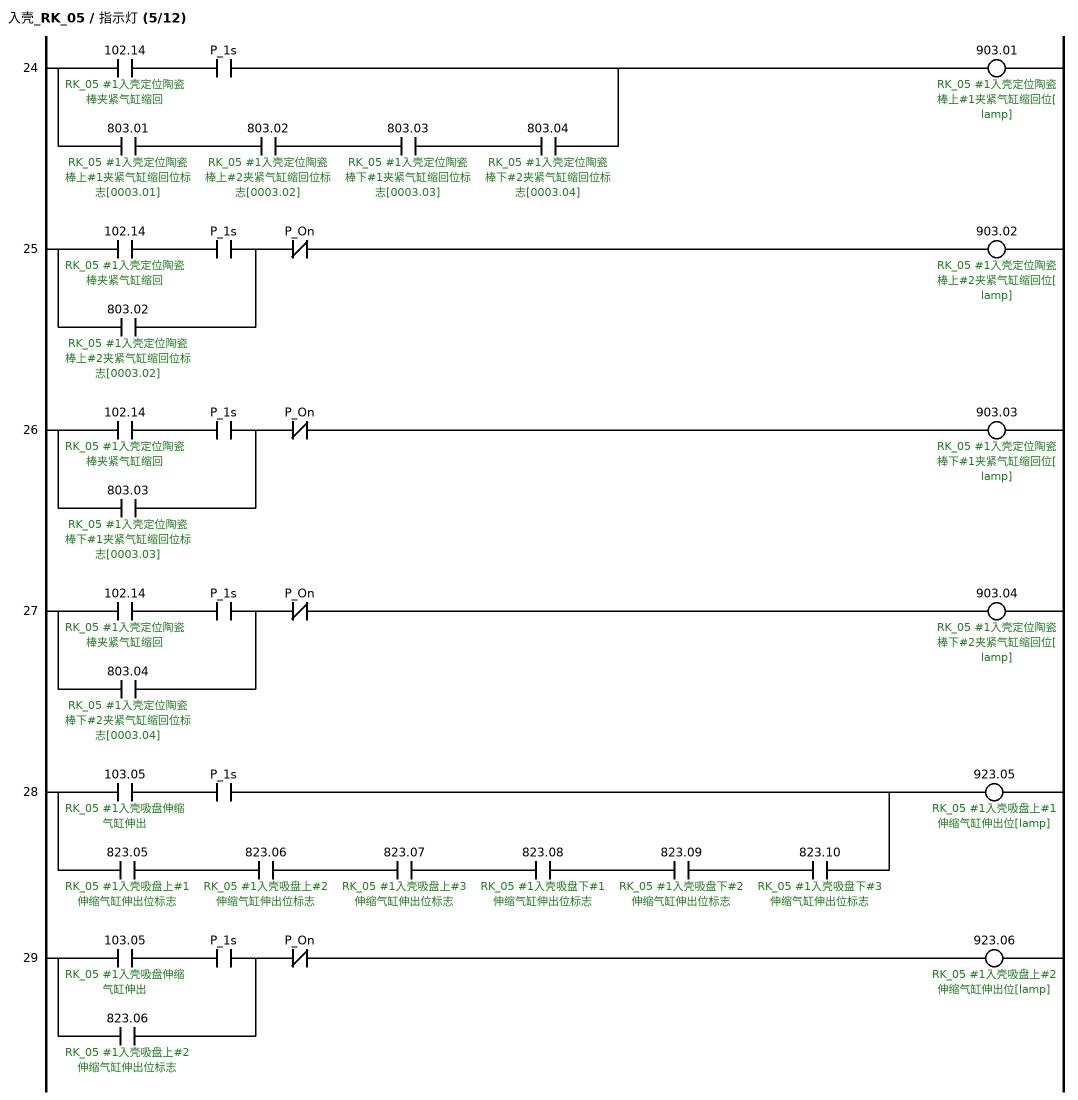
; rung 24
LD 102.14  ; RK_05 #1入壳定位陶瓷棒夹紧气缸缩回
AND P_1s
LD 803.01  ; RK_05 #1入壳定位陶瓷棒上#1夹紧气缸缩回位标志[0003.01]
AND 803.02  ; RK_05 #1入壳定位陶瓷棒上#2夹紧气缸缩回位标志[0003.02]
AND 803.03  ; RK_05 #1入壳定位陶瓷棒下#1夹紧气缸缩回位标志[0003.03]
AND 803.04  ; RK_05 #1入壳定位陶瓷棒下#2夹紧气缸缩回位标志[0003.04]
ORLD
OUT 903.01  ; RK_05 #1入壳定位陶瓷棒上#1夹紧气缸缩回位[lamp]
; rung 25
LD 102.14  ; RK_05 #1入壳定位陶瓷棒夹紧气缸缩回
AND P_1s
OR 803.02  ; RK_05 #1入壳定位陶瓷棒上#2夹紧气缸缩回位标志[0003.02]
ANDNOT P_On
OUT 903.02  ; RK_05 #1入壳定位陶瓷棒上#2夹紧气缸缩回位[lamp]
; rung 26
LD 102.14  ; RK_05 #1入壳定位陶瓷棒夹紧气缸缩回
AND P_1s
OR 803.03  ; RK_05 #1入壳定位陶瓷棒下#1夹紧气缸缩回位标志[0003.03]
ANDNOT P_On
OUT 903.03  ; RK_05 #1入壳定位陶瓷棒下#1夹紧气缸缩回位[lamp]
; rung 27
LD 102.14  ; RK_05 #1入壳定位陶瓷棒夹紧气缸缩回
AND P_1s
OR 803.04  ; RK_05 #1入壳定位陶瓷棒下#2夹紧气缸缩回位标志[0003.04]
ANDNOT P_On
OUT 903.04  ; RK_05 #1入壳定位陶瓷棒下#2夹紧气缸缩回位[lamp]
; rung 28
LD 103.05  ; RK_05 #1入壳吸盘伸缩气缸伸出
AND P_1s
LD 823.05  ; RK_05 #1入壳吸盘上#1伸缩气缸伸出位标志
AND 823.06  ; RK_05 #1入壳吸盘上#2伸缩气缸伸出位标志
AND 823.07  ; RK_05 #1入壳吸盘上#3伸缩气缸伸出位标志
AND 823.08  ; RK_05 #1入壳吸盘下#1伸缩气缸伸出位标志
AND 823.09  ; RK_05 #1入壳吸盘下#2伸缩气缸伸出位标志
AND 823.10  ; RK_05 #1入壳吸盘下#3伸缩气缸伸出位标志
ORLD
OUT 923.05  ; RK_05 #1入壳吸盘上#1伸缩气缸伸出位[lamp]
; rung 29
LD 103.05  ; RK_05 #1入壳吸盘伸缩气缸伸出
AND P_1s
OR 823.06  ; RK_05 #1入壳吸盘上#2伸缩气缸伸出位标志
ANDNOT P_On
OUT 923.06  ; RK_05 #1入壳吸盘上#2伸缩气缸伸出位[lamp]

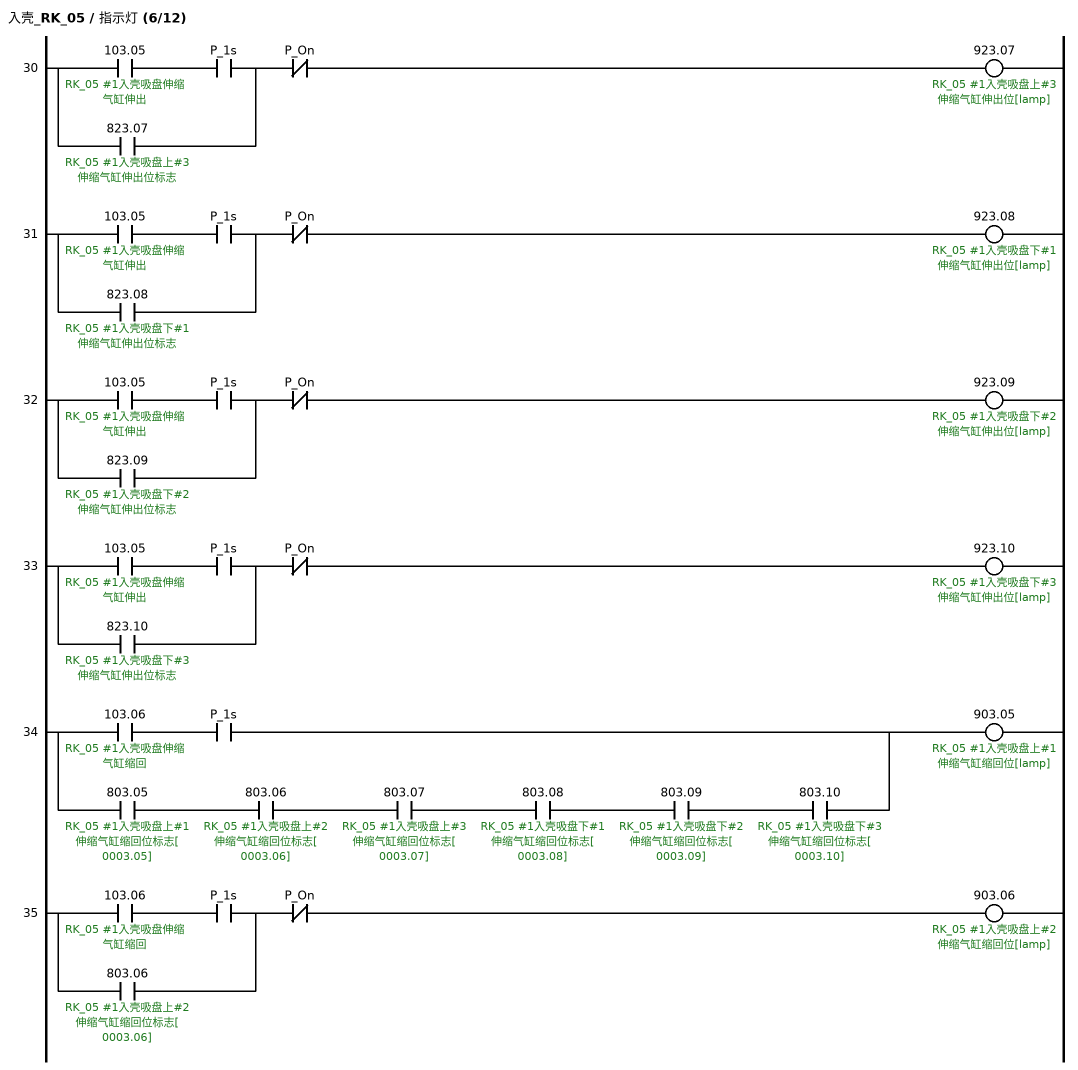
; rung 30
LD 103.05  ; RK_05 #1入壳吸盘伸缩气缸伸出
AND P_1s
OR 823.07  ; RK_05 #1入壳吸盘上#3伸缩气缸伸出位标志
ANDNOT P_On
OUT 923.07  ; RK_05 #1入壳吸盘上#3伸缩气缸伸出位[lamp]
; rung 31
LD 103.05  ; RK_05 #1入壳吸盘伸缩气缸伸出
AND P_1s
OR 823.08  ; RK_05 #1入壳吸盘下#1伸缩气缸伸出位标志
ANDNOT P_On
OUT 923.08  ; RK_05 #1入壳吸盘下#1伸缩气缸伸出位[lamp]
; rung 32
LD 103.05  ; RK_05 #1入壳吸盘伸缩气缸伸出
AND P_1s
OR 823.09  ; RK_05 #1入壳吸盘下#2伸缩气缸伸出位标志
ANDNOT P_On
OUT 923.09  ; RK_05 #1入壳吸盘下#2伸缩气缸伸出位[lamp]
; rung 33
LD 103.05  ; RK_05 #1入壳吸盘伸缩气缸伸出
AND P_1s
OR 823.10  ; RK_05 #1入壳吸盘下#3伸缩气缸伸出位标志
ANDNOT P_On
OUT 923.10  ; RK_05 #1入壳吸盘下#3伸缩气缸伸出位[lamp]
; rung 34
LD 103.06  ; RK_05 #1入壳吸盘伸缩气缸缩回
AND P_1s
LD 803.05  ; RK_05 #1入壳吸盘上#1伸缩气缸缩回位标志[0003.05]
AND 803.06  ; RK_05 #1入壳吸盘上#2伸缩气缸缩回位标志[0003.06]
AND 803.07  ; RK_05 #1入壳吸盘上#3伸缩气缸缩回位标志[0003.07]
AND 803.08  ; RK_05 #1入壳吸盘下#1伸缩气缸缩回位标志[0003.08]
AND 803.09  ; RK_05 #1入壳吸盘下#2伸缩气缸缩回位标志[0003.09]
AND 803.10  ; RK_05 #1入壳吸盘下#3伸缩气缸缩回位标志[0003.10]
ORLD
OUT 903.05  ; RK_05 #1入壳吸盘上#1伸缩气缸缩回位[lamp]
; rung 35
LD 103.06  ; RK_05 #1入壳吸盘伸缩气缸缩回
AND P_1s
OR 803.06  ; RK_05 #1入壳吸盘上#2伸缩气缸缩回位标志[0003.06]
ANDNOT P_On
OUT 903.06  ; RK_05 #1入壳吸盘上#2伸缩气缸缩回位[lamp]

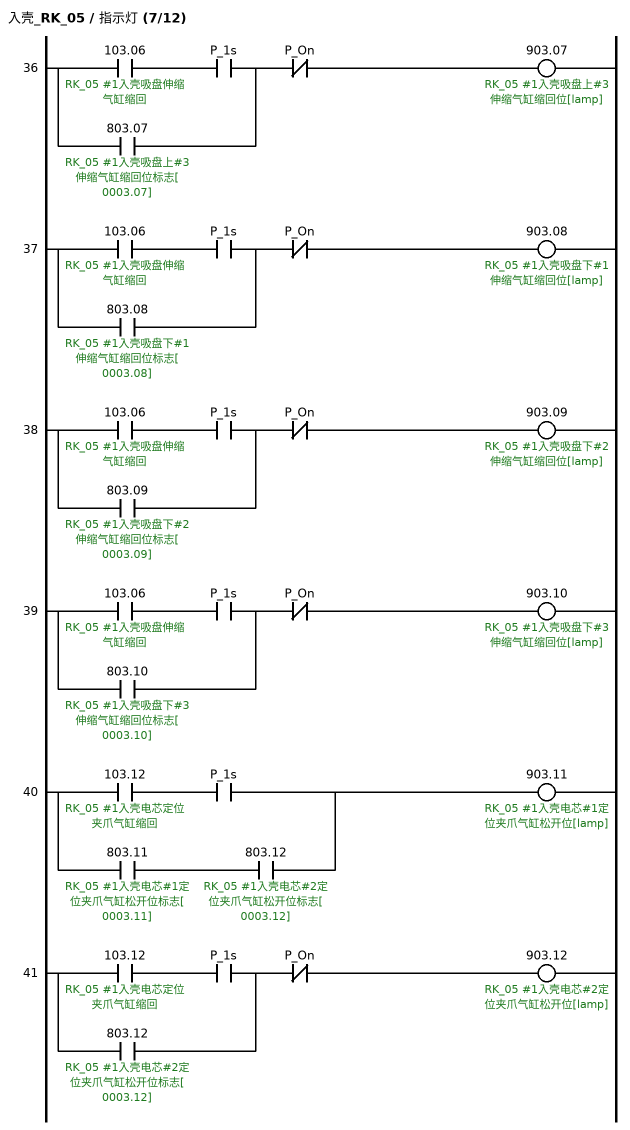
; rung 36
LD 103.06  ; RK_05 #1入壳吸盘伸缩气缸缩回
AND P_1s
OR 803.07  ; RK_05 #1入壳吸盘上#3伸缩气缸缩回位标志[0003.07]
ANDNOT P_On
OUT 903.07  ; RK_05 #1入壳吸盘上#3伸缩气缸缩回位[lamp]
; rung 37
LD 103.06  ; RK_05 #1入壳吸盘伸缩气缸缩回
AND P_1s
OR 803.08  ; RK_05 #1入壳吸盘下#1伸缩气缸缩回位标志[0003.08]
ANDNOT P_On
OUT 903.08  ; RK_05 #1入壳吸盘下#1伸缩气缸缩回位[lamp]
; rung 38
LD 103.06  ; RK_05 #1入壳吸盘伸缩气缸缩回
AND P_1s
OR 803.09  ; RK_05 #1入壳吸盘下#2伸缩气缸缩回位标志[0003.09]
ANDNOT P_On
OUT 903.09  ; RK_05 #1入壳吸盘下#2伸缩气缸缩回位[lamp]
; rung 39
LD 103.06  ; RK_05 #1入壳吸盘伸缩气缸缩回
AND P_1s
OR 803.10  ; RK_05 #1入壳吸盘下#3伸缩气缸缩回位标志[0003.10]
ANDNOT P_On
OUT 903.10  ; RK_05 #1入壳吸盘下#3伸缩气缸缩回位[lamp]
; rung 40
LD 103.12  ; RK_05 #1入壳电芯定位夹爪气缸缩回
AND P_1s
LD 803.11  ; RK_05 #1入壳电芯#1定位夹爪气缸松开位标志[0003.11]
AND 803.12  ; RK_05 #1入壳电芯#2定位夹爪气缸松开位标志[0003.12]
ORLD
OUT 903.11  ; RK_05 #1入壳电芯#1定位夹爪气缸松开位[lamp]
; rung 41
LD 103.12  ; RK_05 #1入壳电芯定位夹爪气缸缩回
AND P_1s
OR 803.12  ; RK_05 #1入壳电芯#2定位夹爪气缸松开位标志[0003.12]
ANDNOT P_On
OUT 903.12  ; RK_05 #1入壳电芯#2定位夹爪气缸松开位[lamp]

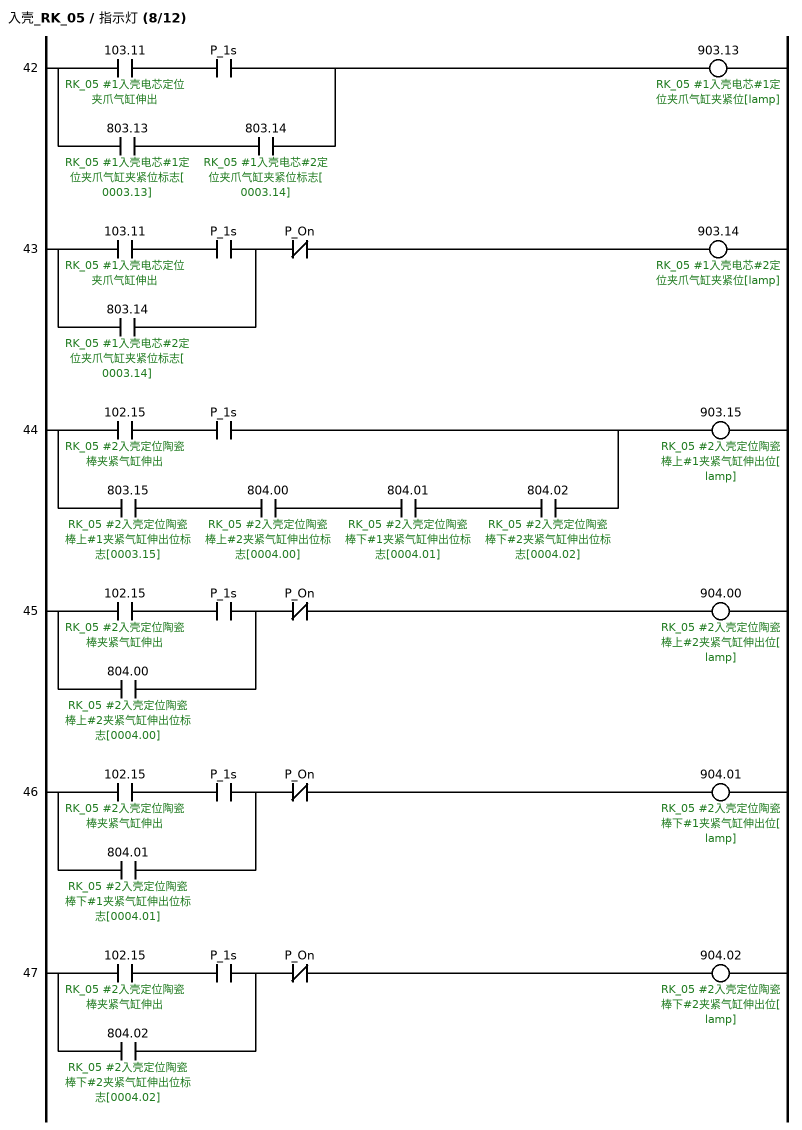
; rung 42
LD 103.11  ; RK_05 #1入壳电芯定位夹爪气缸伸出
AND P_1s
LD 803.13  ; RK_05 #1入壳电芯#1定位夹爪气缸夹紧位标志[0003.13]
AND 803.14  ; RK_05 #1入壳电芯#2定位夹爪气缸夹紧位标志[0003.14]
ORLD
OUT 903.13  ; RK_05 #1入壳电芯#1定位夹爪气缸夹紧位[lamp]
; rung 43
LD 103.11  ; RK_05 #1入壳电芯定位夹爪气缸伸出
AND P_1s
OR 803.14  ; RK_05 #1入壳电芯#2定位夹爪气缸夹紧位标志[0003.14]
ANDNOT P_On
OUT 903.14  ; RK_05 #1入壳电芯#2定位夹爪气缸夹紧位[lamp]
; rung 44
LD 102.15  ; RK_05 #2入壳定位陶瓷棒夹紧气缸伸出
AND P_1s
LD 803.15  ; RK_05 #2入壳定位陶瓷棒上#1夹紧气缸伸出位标志[0003.15]
AND 804.00  ; RK_05 #2入壳定位陶瓷棒上#2夹紧气缸伸出位标志[0004.00]
AND 804.01  ; RK_05 #2入壳定位陶瓷棒下#1夹紧气缸伸出位标志[0004.01]
AND 804.02  ; RK_05 #2入壳定位陶瓷棒下#2夹紧气缸伸出位标志[0004.02]
ORLD
OUT 903.15  ; RK_05 #2入壳定位陶瓷棒上#1夹紧气缸伸出位[lamp]
; rung 45
LD 102.15  ; RK_05 #2入壳定位陶瓷棒夹紧气缸伸出
AND P_1s
OR 804.00  ; RK_05 #2入壳定位陶瓷棒上#2夹紧气缸伸出位标志[0004.00]
ANDNOT P_On
OUT 904.00  ; RK_05 #2入壳定位陶瓷棒上#2夹紧气缸伸出位[lamp]
; rung 46
LD 102.15  ; RK_05 #2入壳定位陶瓷棒夹紧气缸伸出
AND P_1s
OR 804.01  ; RK_05 #2入壳定位陶瓷棒下#1夹紧气缸伸出位标志[0004.01]
ANDNOT P_On
OUT 904.01  ; RK_05 #2入壳定位陶瓷棒下#1夹紧气缸伸出位[lamp]
; rung 47
LD 102.15  ; RK_05 #2入壳定位陶瓷棒夹紧气缸伸出
AND P_1s
OR 804.02  ; RK_05 #2入壳定位陶瓷棒下#2夹紧气缸伸出位标志[0004.02]
ANDNOT P_On
OUT 904.02  ; RK_05 #2入壳定位陶瓷棒下#2夹紧气缸伸出位[lamp]

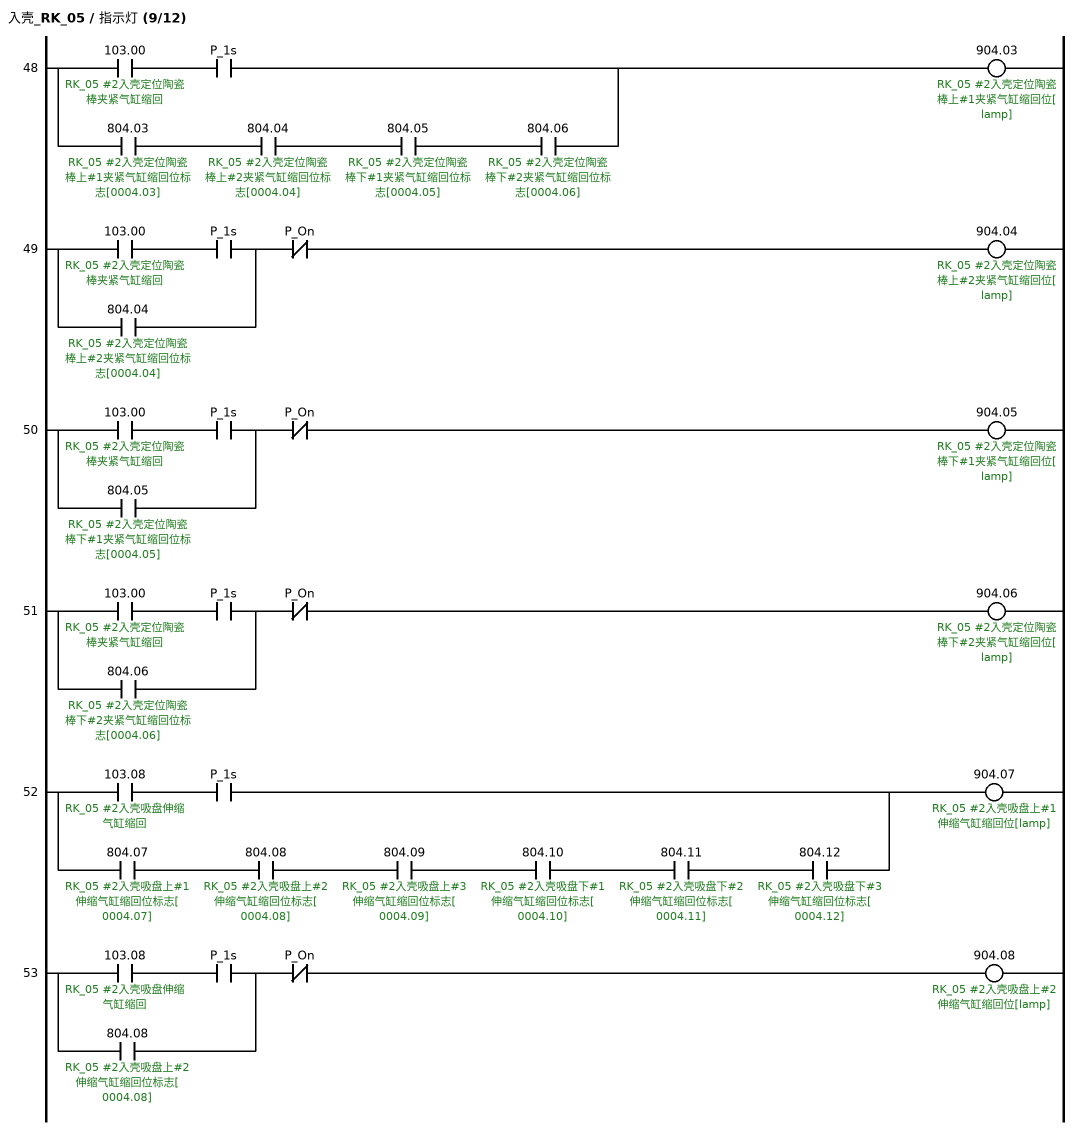
; rung 48
LD 103.00  ; RK_05 #2入壳定位陶瓷棒夹紧气缸缩回
AND P_1s
LD 804.03  ; RK_05 #2入壳定位陶瓷棒上#1夹紧气缸缩回位标志[0004.03]
AND 804.04  ; RK_05 #2入壳定位陶瓷棒上#2夹紧气缸缩回位标志[0004.04]
AND 804.05  ; RK_05 #2入壳定位陶瓷棒下#1夹紧气缸缩回位标志[0004.05]
AND 804.06  ; RK_05 #2入壳定位陶瓷棒下#2夹紧气缸缩回位标志[0004.06]
ORLD
OUT 904.03  ; RK_05 #2入壳定位陶瓷棒上#1夹紧气缸缩回位[lamp]
; rung 49
LD 103.00  ; RK_05 #2入壳定位陶瓷棒夹紧气缸缩回
AND P_1s
OR 804.04  ; RK_05 #2入壳定位陶瓷棒上#2夹紧气缸缩回位标志[0004.04]
ANDNOT P_On
OUT 904.04  ; RK_05 #2入壳定位陶瓷棒上#2夹紧气缸缩回位[lamp]
; rung 50
LD 103.00  ; RK_05 #2入壳定位陶瓷棒夹紧气缸缩回
AND P_1s
OR 804.05  ; RK_05 #2入壳定位陶瓷棒下#1夹紧气缸缩回位标志[0004.05]
ANDNOT P_On
OUT 904.05  ; RK_05 #2入壳定位陶瓷棒下#1夹紧气缸缩回位[lamp]
; rung 51
LD 103.00  ; RK_05 #2入壳定位陶瓷棒夹紧气缸缩回
AND P_1s
OR 804.06  ; RK_05 #2入壳定位陶瓷棒下#2夹紧气缸缩回位标志[0004.06]
ANDNOT P_On
OUT 904.06  ; RK_05 #2入壳定位陶瓷棒下#2夹紧气缸缩回位[lamp]
; rung 52
LD 103.08  ; RK_05 #2入壳吸盘伸缩气缸缩回
AND P_1s
LD 804.07  ; RK_05 #2入壳吸盘上#1伸缩气缸缩回位标志[0004.07]
AND 804.08  ; RK_05 #2入壳吸盘上#2伸缩气缸缩回位标志[0004.08]
AND 804.09  ; RK_05 #2入壳吸盘上#3伸缩气缸缩回位标志[0004.09]
AND 804.10  ; RK_05 #2入壳吸盘下#1伸缩气缸缩回位标志[0004.10]
AND 804.11  ; RK_05 #2入壳吸盘下#2伸缩气缸缩回位标志[0004.11]
AND 804.12  ; RK_05 #2入壳吸盘下#3伸缩气缸缩回位标志[0004.12]
ORLD
OUT 904.07  ; RK_05 #2入壳吸盘上#1伸缩气缸缩回位[lamp]
; rung 53
LD 103.08  ; RK_05 #2入壳吸盘伸缩气缸缩回
AND P_1s
OR 804.08  ; RK_05 #2入壳吸盘上#2伸缩气缸缩回位标志[0004.08]
ANDNOT P_On
OUT 904.08  ; RK_05 #2入壳吸盘上#2伸缩气缸缩回位[lamp]

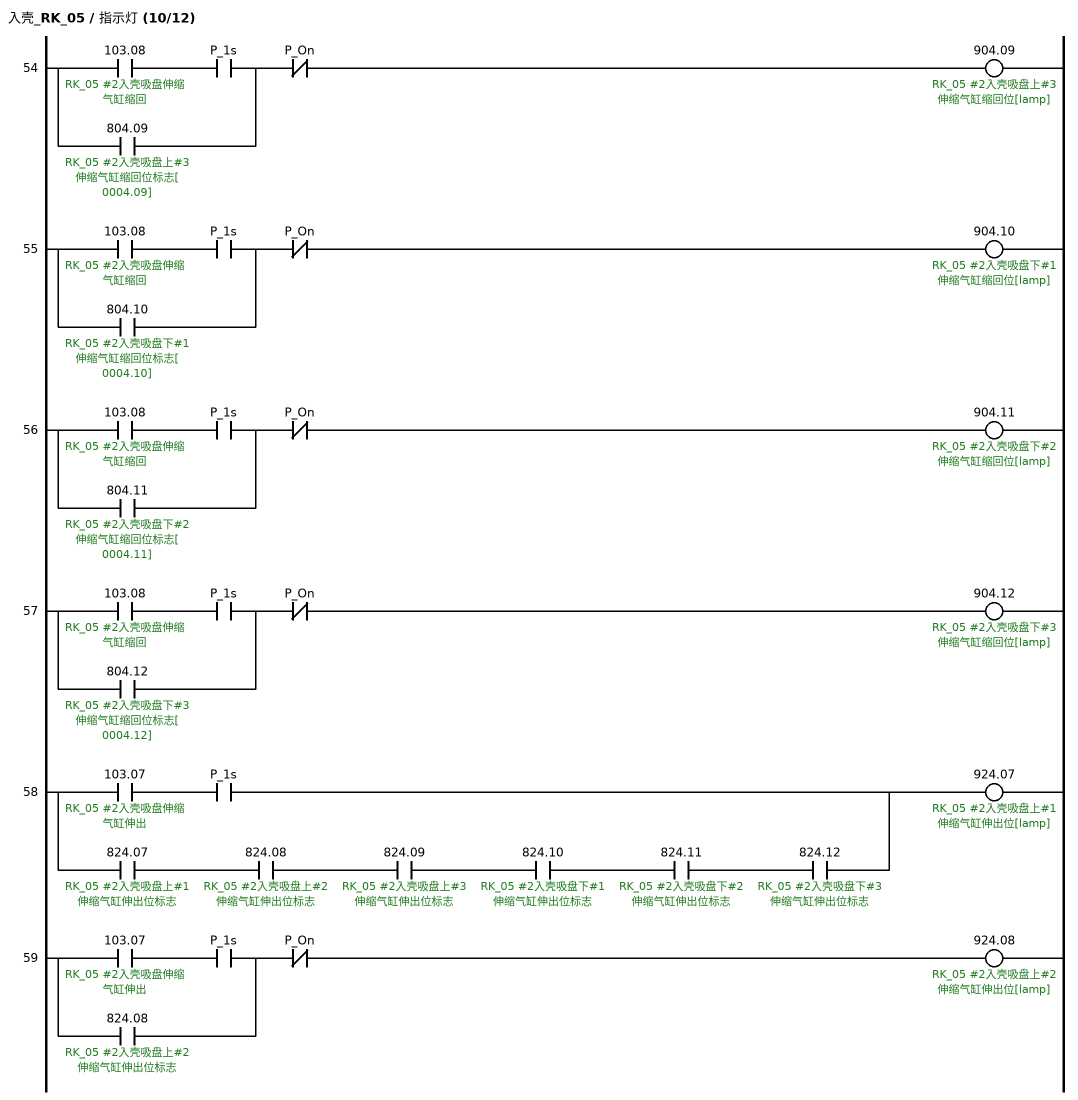
; rung 54
LD 103.08  ; RK_05 #2入壳吸盘伸缩气缸缩回
AND P_1s
OR 804.09  ; RK_05 #2入壳吸盘上#3伸缩气缸缩回位标志[0004.09]
ANDNOT P_On
OUT 904.09  ; RK_05 #2入壳吸盘上#3伸缩气缸缩回位[lamp]
; rung 55
LD 103.08  ; RK_05 #2入壳吸盘伸缩气缸缩回
AND P_1s
OR 804.10  ; RK_05 #2入壳吸盘下#1伸缩气缸缩回位标志[0004.10]
ANDNOT P_On
OUT 904.10  ; RK_05 #2入壳吸盘下#1伸缩气缸缩回位[lamp]
; rung 56
LD 103.08  ; RK_05 #2入壳吸盘伸缩气缸缩回
AND P_1s
OR 804.11  ; RK_05 #2入壳吸盘下#2伸缩气缸缩回位标志[0004.11]
ANDNOT P_On
OUT 904.11  ; RK_05 #2入壳吸盘下#2伸缩气缸缩回位[lamp]
; rung 57
LD 103.08  ; RK_05 #2入壳吸盘伸缩气缸缩回
AND P_1s
OR 804.12  ; RK_05 #2入壳吸盘下#3伸缩气缸缩回位标志[0004.12]
ANDNOT P_On
OUT 904.12  ; RK_05 #2入壳吸盘下#3伸缩气缸缩回位[lamp]
; rung 58
LD 103.07  ; RK_05 #2入壳吸盘伸缩气缸伸出
AND P_1s
LD 824.07  ; RK_05 #2入壳吸盘上#1伸缩气缸伸出位标志
AND 824.08  ; RK_05 #2入壳吸盘上#2伸缩气缸伸出位标志
AND 824.09  ; RK_05 #2入壳吸盘上#3伸缩气缸伸出位标志
AND 824.10  ; RK_05 #2入壳吸盘下#1伸缩气缸伸出位标志
AND 824.11  ; RK_05 #2入壳吸盘下#2伸缩气缸伸出位标志
AND 824.12  ; RK_05 #2入壳吸盘下#3伸缩气缸伸出位标志
ORLD
OUT 924.07  ; RK_05 #2入壳吸盘上#1伸缩气缸伸出位[lamp]
; rung 59
LD 103.07  ; RK_05 #2入壳吸盘伸缩气缸伸出
AND P_1s
OR 824.08  ; RK_05 #2入壳吸盘上#2伸缩气缸伸出位标志
ANDNOT P_On
OUT 924.08  ; RK_05 #2入壳吸盘上#2伸缩气缸伸出位[lamp]

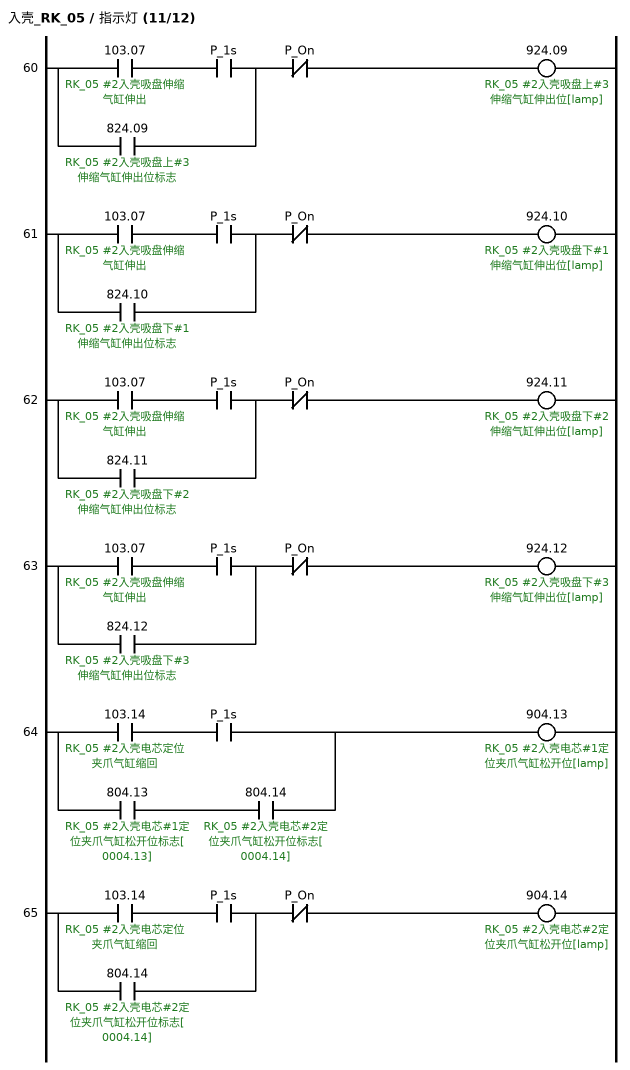
; rung 60
LD 103.07  ; RK_05 #2入壳吸盘伸缩气缸伸出
AND P_1s
OR 824.09  ; RK_05 #2入壳吸盘上#3伸缩气缸伸出位标志
ANDNOT P_On
OUT 924.09  ; RK_05 #2入壳吸盘上#3伸缩气缸伸出位[lamp]
; rung 61
LD 103.07  ; RK_05 #2入壳吸盘伸缩气缸伸出
AND P_1s
OR 824.10  ; RK_05 #2入壳吸盘下#1伸缩气缸伸出位标志
ANDNOT P_On
OUT 924.10  ; RK_05 #2入壳吸盘下#1伸缩气缸伸出位[lamp]
; rung 62
LD 103.07  ; RK_05 #2入壳吸盘伸缩气缸伸出
AND P_1s
OR 824.11  ; RK_05 #2入壳吸盘下#2伸缩气缸伸出位标志
ANDNOT P_On
OUT 924.11  ; RK_05 #2入壳吸盘下#2伸缩气缸伸出位[lamp]
; rung 63
LD 103.07  ; RK_05 #2入壳吸盘伸缩气缸伸出
AND P_1s
OR 824.12  ; RK_05 #2入壳吸盘下#3伸缩气缸伸出位标志
ANDNOT P_On
OUT 924.12  ; RK_05 #2入壳吸盘下#3伸缩气缸伸出位[lamp]
; rung 64
LD 103.14  ; RK_05 #2入壳电芯定位夹爪气缸缩回
AND P_1s
LD 804.13  ; RK_05 #2入壳电芯#1定位夹爪气缸松开位标志[0004.13]
AND 804.14  ; RK_05 #2入壳电芯#2定位夹爪气缸松开位标志[0004.14]
ORLD
OUT 904.13  ; RK_05 #2入壳电芯#1定位夹爪气缸松开位[lamp]
; rung 65
LD 103.14  ; RK_05 #2入壳电芯定位夹爪气缸缩回
AND P_1s
OR 804.14  ; RK_05 #2入壳电芯#2定位夹爪气缸松开位标志[0004.14]
ANDNOT P_On
OUT 904.14  ; RK_05 #2入壳电芯#2定位夹爪气缸松开位[lamp]

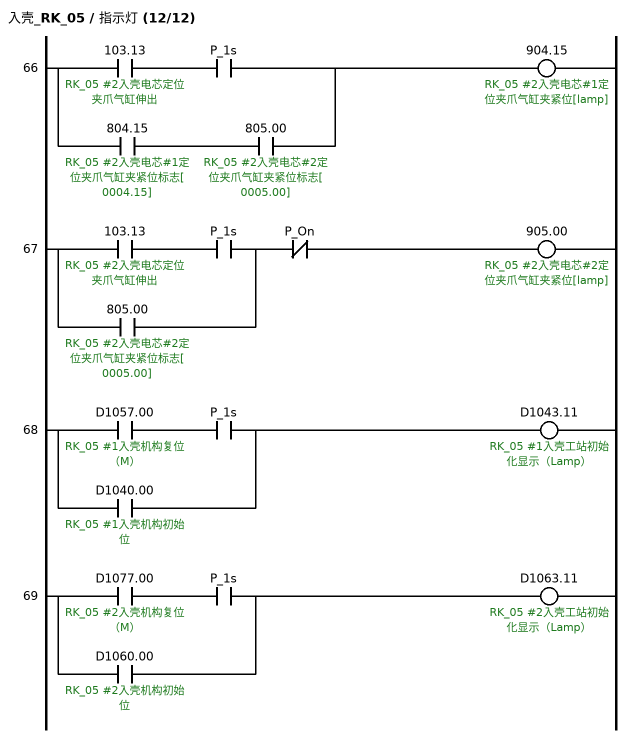
; rung 66
LD 103.13  ; RK_05 #2入壳电芯定位夹爪气缸伸出
AND P_1s
LD 804.15  ; RK_05 #2入壳电芯#1定位夹爪气缸夹紧位标志[0004.15]
AND 805.00  ; RK_05 #2入壳电芯#2定位夹爪气缸夹紧位标志[0005.00]
ORLD
OUT 904.15  ; RK_05 #2入壳电芯#1定位夹爪气缸夹紧位[lamp]
; rung 67
LD 103.13  ; RK_05 #2入壳电芯定位夹爪气缸伸出
AND P_1s
OR 805.00  ; RK_05 #2入壳电芯#2定位夹爪气缸夹紧位标志[0005.00]
ANDNOT P_On
OUT 905.00  ; RK_05 #2入壳电芯#2定位夹爪气缸夹紧位[lamp]
; rung 68
LD D1057.00  ; RK_05 #1入壳机构复位（M）
AND P_1s
OR D1040.00  ; RK_05 #1入壳机构初始位
OUT D1043.11  ; RK_05 #1入壳工站初始化显示（Lamp）
; rung 69
LD D1077.00  ; RK_05 #2入壳机构复位（M）
AND P_1s
OR D1060.00  ; RK_05 #2入壳机构初始位
OUT D1063.11  ; RK_05 #2入壳工站初始化显示（Lamp）

### Section 外部输出

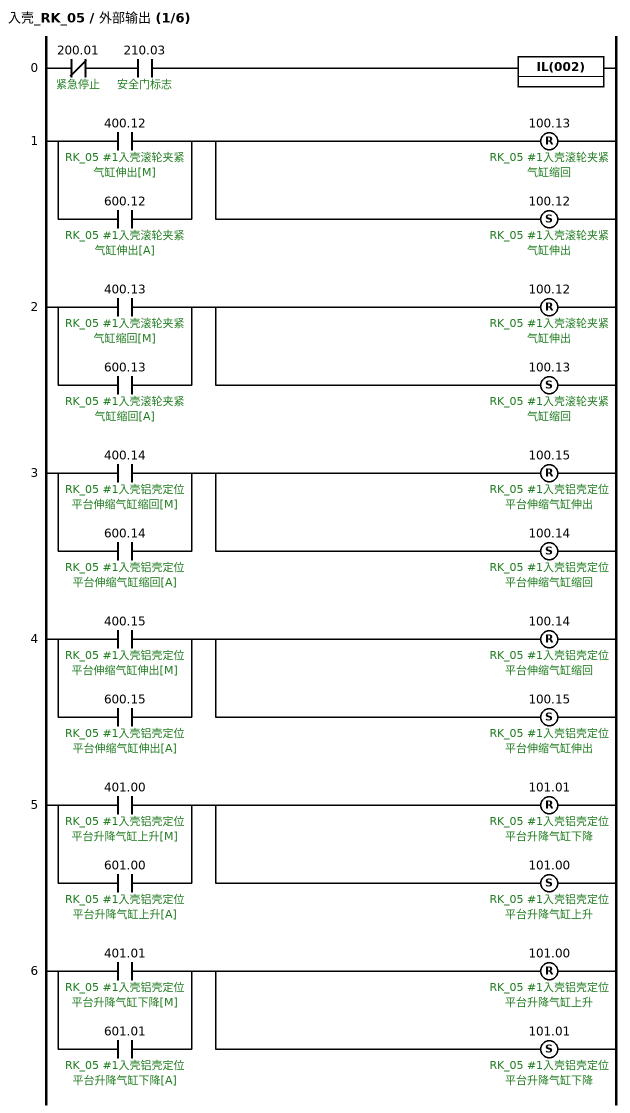
; rung 0
LDNOT 200.01  ; 紧急停止
AND 210.03  ; 安全门标志
IL(002)
; rung 1
LD 400.12  ; RK_05 #1入壳滚轮夹紧气缸伸出[M]
OR 600.12  ; RK_05 #1入壳滚轮夹紧气缸伸出[A]
RSET 100.13  ; RK_05 #1入壳滚轮夹紧气缸缩回
SET 100.12  ; RK_05 #1入壳滚轮夹紧气缸伸出
; rung 2
LD 400.13  ; RK_05 #1入壳滚轮夹紧气缸缩回[M]
OR 600.13  ; RK_05 #1入壳滚轮夹紧气缸缩回[A]
RSET 100.12  ; RK_05 #1入壳滚轮夹紧气缸伸出
SET 100.13  ; RK_05 #1入壳滚轮夹紧气缸缩回
; rung 3
LD 400.14  ; RK_05 #1入壳铝壳定位平台伸缩气缸缩回[M]
OR 600.14  ; RK_05 #1入壳铝壳定位平台伸缩气缸缩回[A]
RSET 100.15  ; RK_05 #1入壳铝壳定位平台伸缩气缸伸出
SET 100.14  ; RK_05 #1入壳铝壳定位平台伸缩气缸缩回
; rung 4
LD 400.15  ; RK_05 #1入壳铝壳定位平台伸缩气缸伸出[M]
OR 600.15  ; RK_05 #1入壳铝壳定位平台伸缩气缸伸出[A]
RSET 100.14  ; RK_05 #1入壳铝壳定位平台伸缩气缸缩回
SET 100.15  ; RK_05 #1入壳铝壳定位平台伸缩气缸伸出
; rung 5
LD 401.00  ; RK_05 #1入壳铝壳定位平台升降气缸上升[M]
OR 601.00  ; RK_05 #1入壳铝壳定位平台升降气缸上升[A]
RSET 101.01  ; RK_05 #1入壳铝壳定位平台升降气缸下降
SET 101.00  ; RK_05 #1入壳铝壳定位平台升降气缸上升
; rung 6
LD 401.01  ; RK_05 #1入壳铝壳定位平台升降气缸下降[M]
OR 601.01  ; RK_05 #1入壳铝壳定位平台升降气缸下降[A]
RSET 101.00  ; RK_05 #1入壳铝壳定位平台升降气缸上升
SET 101.01  ; RK_05 #1入壳铝壳定位平台升降气缸下降

